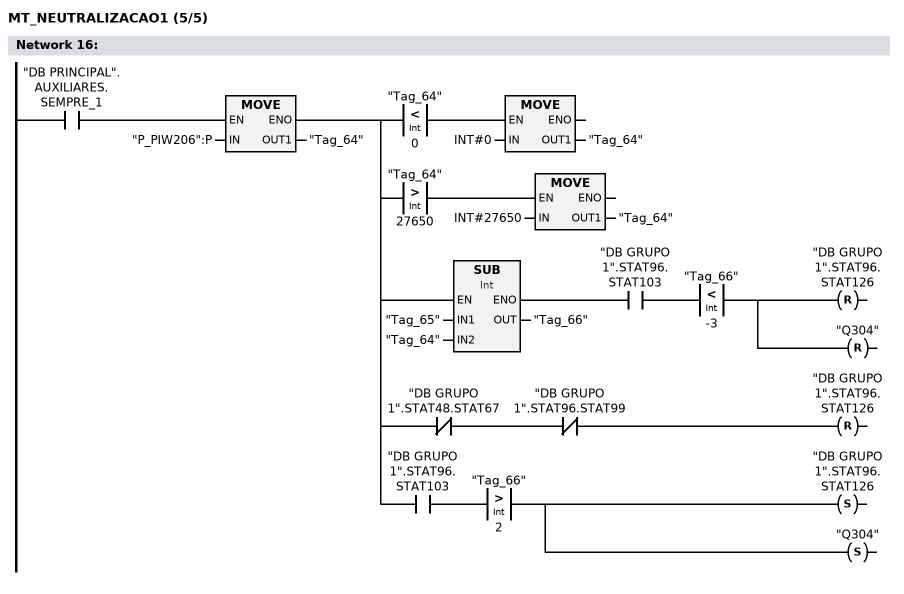
   RUNG wire#powerrail
      Contact( "DB PRINCIPAL".AUXILIARES.SEMPRE_1 )
      { S7_GenerateENO := "TRUE" } Move(in := "P_PIW206":P, out1 => "Tag_64")
      wire#w1
      { S7_Templates := "SrcType := Int" } LT_Contact(in1 := "Tag_64", in2 := 0)
      { S7_GenerateENO := "TRUE" } Move(in := INT#0, out1 => "Tag_64")
   END_RUNG
   RUNG wire#w1
      { S7_Templates := "SrcType := Int" } GT_Contact(in1 := "Tag_64", in2 := 27650)
      { S7_GenerateENO := "TRUE" } Move(in := INT#27650, out1 => "Tag_64")
   END_RUNG
   RUNG wire#w1
      { S7_Templates := "SrcType := Int"; S7_GenerateENO := "TRUE" } Sub(in1 := "Tag_65", in2 := "Tag_64", out => "Tag_66")
      Contact( "DB GRUPO 1".STAT96.STAT103 )
      { S7_Templates := "SrcType := Int" } LT_Contact(in1 := "Tag_66", in2 := -3)
      wire#w2
      R_Coil( "DB GRUPO 1".STAT96.STAT126 )
   END_RUNG
   RUNG wire#w2
      R_Coil( "Q304" )
   END_RUNG
   RUNG wire#w1
      I_Contact( "DB GRUPO 1".STAT48.STAT67 )
      I_Contact( "DB GRUPO 1".STAT96.STAT99 )
      R_Coil( "DB GRUPO 1".STAT96.STAT126 )
   END_RUNG
   RUNG wire#w1
      Contact( "DB GRUPO 1".STAT96.STAT103 )
      { S7_Templates := "SrcType := Int" } GT_Contact(in1 := "Tag_66", in2 := 2)
      wire#w3
      S_Coil( "DB GRUPO 1".STAT96.STAT126 )
   END_RUNG
   RUNG wire#w3
      S_Coil( "Q304" )
   END_RUNG
   // the same network as SCL:
   // ENO of a box is taken as its EN; it also drops when the box reports an error
   IF "DB PRINCIPAL".AUXILIARES.SEMPRE_1 THEN "Tag_64" := "P_PIW206":P; END_IF;
   IF "DB PRINCIPAL".AUXILIARES.SEMPRE_1 AND ("Tag_64" < 0) THEN "Tag_64" := INT#0; END_IF;
   IF "DB PRINCIPAL".AUXILIARES.SEMPRE_1 AND ("Tag_64" > 27650) THEN "Tag_64" := INT#27650; END_IF;
   IF "DB PRINCIPAL".AUXILIARES.SEMPRE_1 THEN "Tag_66" := "Tag_65" - "Tag_64"; END_IF;
   IF "DB PRINCIPAL".AUXILIARES.SEMPRE_1 AND "DB GRUPO 1".STAT96.STAT103 AND ("Tag_66" < (-3)) THEN
       "DB GRUPO 1".STAT96.STAT126 := FALSE;
       "Q304" := FALSE;
   END_IF;
   IF "DB PRINCIPAL".AUXILIARES.SEMPRE_1 AND NOT "DB GRUPO 1".STAT48.STAT67 AND NOT "DB GRUPO 1".STAT96.STAT99 THEN
       "DB GRUPO 1".STAT96.STAT126 := FALSE;
   END_IF;
   IF "DB PRINCIPAL".AUXILIARES.SEMPRE_1 AND "DB GRUPO 1".STAT96.STAT103 AND ("Tag_66" > 2) THEN
       "DB GRUPO 1".STAT96.STAT126 := TRUE;
       "Q304" := TRUE;
   END_IF;
END_REGION
END_FUNCTION

FUNCTION "MT_EXTRACTA1" : Void   // FC13, LAD
TITLE = MÓDULO DE CONTROLE DA EXTRACTA 1
{ S7_Optimized_Access := 'FALSE' }
AUTHOR : THALLES
FAMILY : TRAÇÃO
NAME : LINHA1
VERSION : 0.1
// DATA BLOCK DE CONTROLE // DB13
// Automation Pack Automação Indl. e Com. Ltda.
// Cliente: Texima S/A Ind. de Máquinas
// Cliente Final: Cia. Fiação e Tecidos Santo Antonio.
// Máquina: Sanforizadeira SMT-15 - O.S.: 24.626
   VAR_TEMP
      AUX_R : Real;
   END_VAR
   VAR_TEMP   // added for the SCL form of the ladder/FBD networks
      _w1 : Bool;
      _w2 : Bool;
   END_VAR
BEGIN

REGION Network 1: ALARMES
   // RESET DOS ALARMES
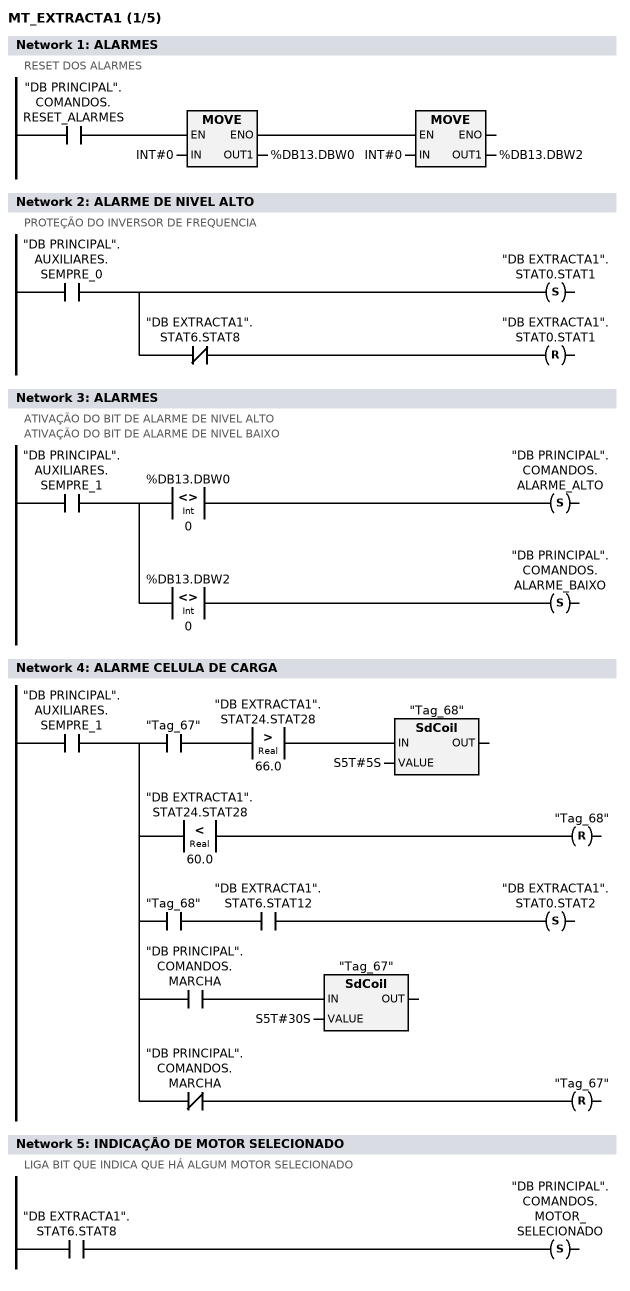
   RUNG wire#powerrail
      Contact( "DB PRINCIPAL".COMANDOS.RESET_ALARMES )
      { S7_GenerateENO := "TRUE" } Move(in := INT#0, out1 => %DB13.DBW0)
      { S7_GenerateENO := "TRUE" } Move(in := INT#0, out1 => %DB13.DBW2)
   END_RUNG
   // the same network as SCL:
   // ENO of a box is taken as its EN; it also drops when the box reports an error
   IF "DB PRINCIPAL".COMANDOS.RESET_ALARMES THEN
       %DB13.DBW0 := INT#0;
       %DB13.DBW2 := INT#0;
   END_IF;
END_REGION

REGION Network 2: ALARME DE NIVEL ALTO
   // PROTEÇÃO DO INVERSOR DE FREQUENCIA
   RUNG wire#powerrail
      Contact( "DB PRINCIPAL".AUXILIARES.SEMPRE_0 )
      wire#w1
      S_Coil( "DB EXTRACTA1".STAT0.STAT1 )
   END_RUNG
   RUNG wire#w1
      I_Contact( "DB EXTRACTA1".STAT6.STAT8 )
      R_Coil( "DB EXTRACTA1".STAT0.STAT1 )
   END_RUNG
   // the same network as SCL:
   IF "DB PRINCIPAL".AUXILIARES.SEMPRE_0 THEN "DB EXTRACTA1".STAT0.STAT1 := TRUE; END_IF;
   IF "DB PRINCIPAL".AUXILIARES.SEMPRE_0 AND NOT "DB EXTRACTA1".STAT6.STAT8 THEN
       "DB EXTRACTA1".STAT0.STAT1 := FALSE;
   END_IF;
END_REGION

REGION Network 3: ALARMES
   // ATIVAÇÃO DO BIT DE ALARME DE NIVEL ALTO
   // ATIVAÇÃO DO BIT DE ALARME DE NIVEL BAIXO
   RUNG wire#powerrail
      Contact( "DB PRINCIPAL".AUXILIARES.SEMPRE_1 )
      wire#w1
      { S7_Templates := "SrcType := Int" } NE_Contact(in1 := %DB13.DBW0, in2 := 0)
      S_Coil( "DB PRINCIPAL".COMANDOS.ALARME_ALTO )
   END_RUNG
   RUNG wire#w1
      { S7_Templates := "SrcType := Int" } NE_Contact(in1 := %DB13.DBW2, in2 := 0)
      S_Coil( "DB PRINCIPAL".COMANDOS.ALARME_BAIXO )
   END_RUNG
   // the same network as SCL:
   IF "DB PRINCIPAL".AUXILIARES.SEMPRE_1 AND (%DB13.DBW0 <> 0) THEN
       "DB PRINCIPAL".COMANDOS.ALARME_ALTO := TRUE;
   END_IF;
   IF "DB PRINCIPAL".AUXILIARES.SEMPRE_1 AND (%DB13.DBW2 <> 0) THEN
       "DB PRINCIPAL".COMANDOS.ALARME_BAIXO := TRUE;
   END_IF;
END_REGION

REGION Network 4: ALARME CELULA DE CARGA
   // no SCL statement known for SdCoil: written as a call
   #_w1 := "DB PRINCIPAL".AUXILIARES.SEMPRE_1;
   SdCoil(value := S5T#5S,
          in := "DB PRINCIPAL".AUXILIARES.SEMPRE_1 AND "Tag_67" AND ("DB EXTRACTA1".STAT24.STAT28 > 66.0),
          operand := "Tag_68");
   IF #_w1 AND ("DB EXTRACTA1".STAT24.STAT28 < 60.0) THEN "Tag_68" := FALSE; END_IF;
   IF #_w1 AND "Tag_68" AND "DB EXTRACTA1".STAT6.STAT12 THEN "DB EXTRACTA1".STAT0.STAT2 := TRUE; END_IF;
   SdCoil(value := S5T#30S, operand := "Tag_67", in := #_w1 AND "DB PRINCIPAL".COMANDOS.MARCHA);
   IF #_w1 AND NOT "DB PRINCIPAL".COMANDOS.MARCHA THEN "Tag_67" := FALSE; END_IF;
END_REGION

REGION Network 5: INDICAÇÃO DE MOTOR SELECIONADO
   // LIGA BIT QUE INDICA QUE HÁ ALGUM MOTOR SELECIONADO
   RUNG wire#powerrail
      Contact( "DB EXTRACTA1".STAT6.STAT8 )
      S_Coil( "DB PRINCIPAL".COMANDOS.MOTOR_SELECIONADO )
   END_RUNG
   // the same network as SCL:
   IF "DB EXTRACTA1".STAT6.STAT8 THEN "DB PRINCIPAL".COMANDOS.MOTOR_SELECIONADO := TRUE; END_IF;
END_REGION

REGION Network 6: COMANDO PARA SELEÇÃO DO MOTOR
   // COMANDO PARA SELEÇÃO DO MOTOR
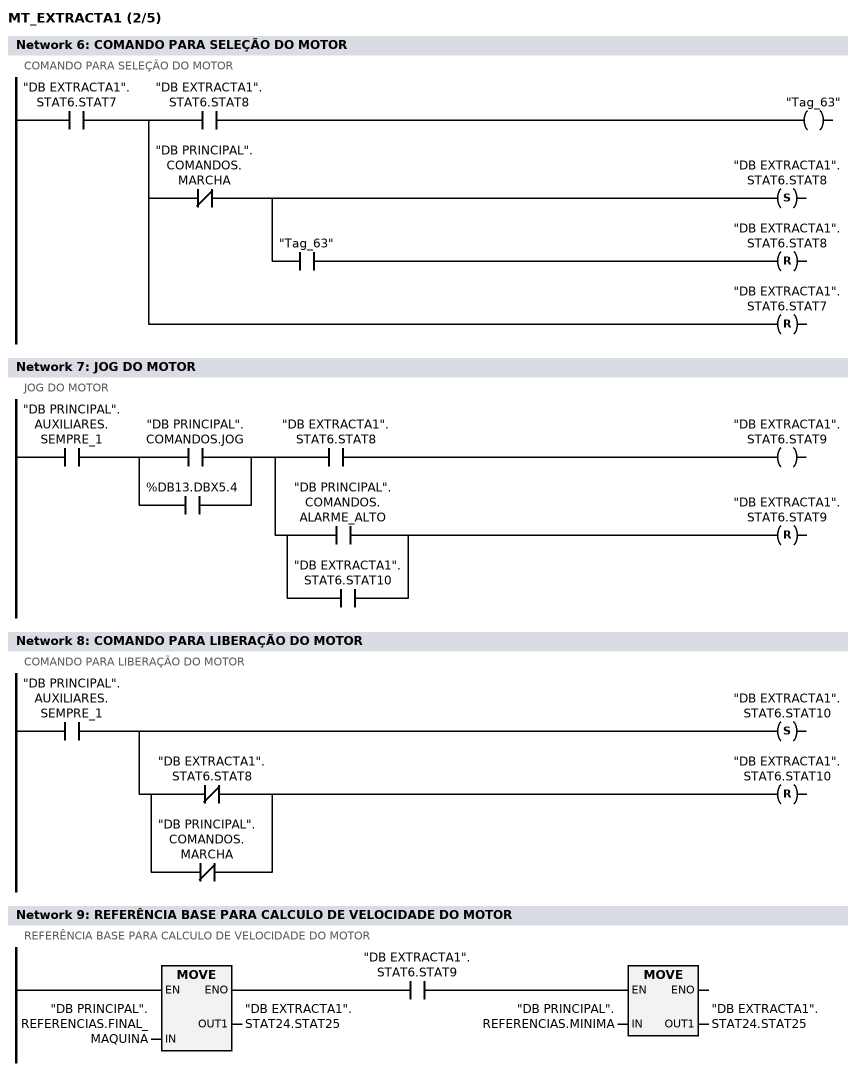
   RUNG wire#powerrail
      Contact( "DB EXTRACTA1".STAT6.STAT7 )
      wire#w1
      Contact( "DB EXTRACTA1".STAT6.STAT8 )
      Coil( "Tag_63" )
   END_RUNG
   RUNG wire#w1
      I_Contact( "DB PRINCIPAL".COMANDOS.MARCHA )
      wire#w2
      S_Coil( "DB EXTRACTA1".STAT6.STAT8 )
   END_RUNG
   RUNG wire#w2
      Contact( "Tag_63" )
      R_Coil( "DB EXTRACTA1".STAT6.STAT8 )
   END_RUNG
   RUNG wire#w1
      R_Coil( "DB EXTRACTA1".STAT6.STAT7 )
   END_RUNG
   // the same network as SCL:
   "Tag_63" := "DB EXTRACTA1".STAT6.STAT7 AND "DB EXTRACTA1".STAT6.STAT8;
   #_w1 := "DB EXTRACTA1".STAT6.STAT7 AND NOT "DB PRINCIPAL".COMANDOS.MARCHA;
   IF #_w1 THEN "DB EXTRACTA1".STAT6.STAT8 := TRUE; END_IF;
   IF #_w1 AND "Tag_63" THEN "DB EXTRACTA1".STAT6.STAT8 := FALSE; END_IF;
   IF "DB EXTRACTA1".STAT6.STAT7 THEN "DB EXTRACTA1".STAT6.STAT7 := FALSE; END_IF;
END_REGION

REGION Network 7: JOG DO MOTOR
   // JOG DO MOTOR
   RUNG wire#powerrail
      Contact( "DB PRINCIPAL".AUXILIARES.SEMPRE_1 )
      wire#w1
      Contact( "DB PRINCIPAL".COMANDOS.JOG )
      wire#w2
      Contact( "DB EXTRACTA1".STAT6.STAT8 )
      Coil( "DB EXTRACTA1".STAT6.STAT9 )
   END_RUNG
   RUNG wire#w1
      Contact( %DB13.DBX5.4 )
   END_RUNG wire#w2
   RUNG wire#w2
      Contact( "DB PRINCIPAL".COMANDOS.ALARME_ALTO )
      wire#w3
      R_Coil( "DB EXTRACTA1".STAT6.STAT9 )
   END_RUNG
   RUNG wire#w2
      Contact( "DB EXTRACTA1".STAT6.STAT10 )
   END_RUNG wire#w3
   // the same network as SCL:
   #_w1 := "DB PRINCIPAL".AUXILIARES.SEMPRE_1 AND ("DB PRINCIPAL".COMANDOS.JOG OR %DB13.DBX5.4);
   "DB EXTRACTA1".STAT6.STAT9 := #_w1 AND "DB EXTRACTA1".STAT6.STAT8;
   IF #_w1 AND ("DB PRINCIPAL".COMANDOS.ALARME_ALTO OR "DB EXTRACTA1".STAT6.STAT10) THEN
       "DB EXTRACTA1".STAT6.STAT9 := FALSE;
   END_IF;
END_REGION

REGION Network 8: COMANDO PARA LIBERAÇÃO DO MOTOR
   // COMANDO PARA LIBERAÇÃO DO MOTOR
   RUNG wire#powerrail
      Contact( "DB PRINCIPAL".AUXILIARES.SEMPRE_1 )
      wire#w1
      S_Coil( "DB EXTRACTA1".STAT6.STAT10 )
   END_RUNG
   RUNG wire#w1
      I_Contact( "DB EXTRACTA1".STAT6.STAT8 )
      wire#w2
      R_Coil( "DB EXTRACTA1".STAT6.STAT10 )
   END_RUNG
   RUNG wire#w1
      I_Contact( "DB PRINCIPAL".COMANDOS.MARCHA )
   END_RUNG wire#w2
   // the same network as SCL:
   IF "DB PRINCIPAL".AUXILIARES.SEMPRE_1 THEN "DB EXTRACTA1".STAT6.STAT10 := TRUE; END_IF;
   IF "DB PRINCIPAL".AUXILIARES.SEMPRE_1 AND (NOT "DB EXTRACTA1".STAT6.STAT8 OR NOT "DB PRINCIPAL".COMANDOS.MARCHA) THEN
       "DB EXTRACTA1".STAT6.STAT10 := FALSE;
   END_IF;
END_REGION

REGION Network 9: REFERÊNCIA BASE PARA CALCULO DE VELOCIDADE DO MOTOR
   // REFERÊNCIA BASE PARA CALCULO DE VELOCIDADE DO MOTOR
   RUNG wire#powerrail
      { S7_GenerateENO := "TRUE" } Move(in := "DB PRINCIPAL".REFERENCIAS.FINAL_MAQUINA, out1 => "DB EXTRACTA1".STAT24.STAT25)
      Contact( "DB EXTRACTA1".STAT6.STAT9 )
      { S7_GenerateENO := "TRUE" } Move(in := "DB PRINCIPAL".REFERENCIAS.MINIMA, out1 => "DB EXTRACTA1".STAT24.STAT25)
   END_RUNG
   // the same network as SCL:
   // ENO of a box is taken as its EN; it also drops when the box reports an error
   "DB EXTRACTA1".STAT24.STAT25 := "DB PRINCIPAL".REFERENCIAS.FINAL_MAQUINA;
   IF "DB EXTRACTA1".STAT6.STAT9 THEN
       "DB EXTRACTA1".STAT24.STAT25 := "DB PRINCIPAL".REFERENCIAS.MINIMA;
   END_IF;
END_REGION

REGION Network 10
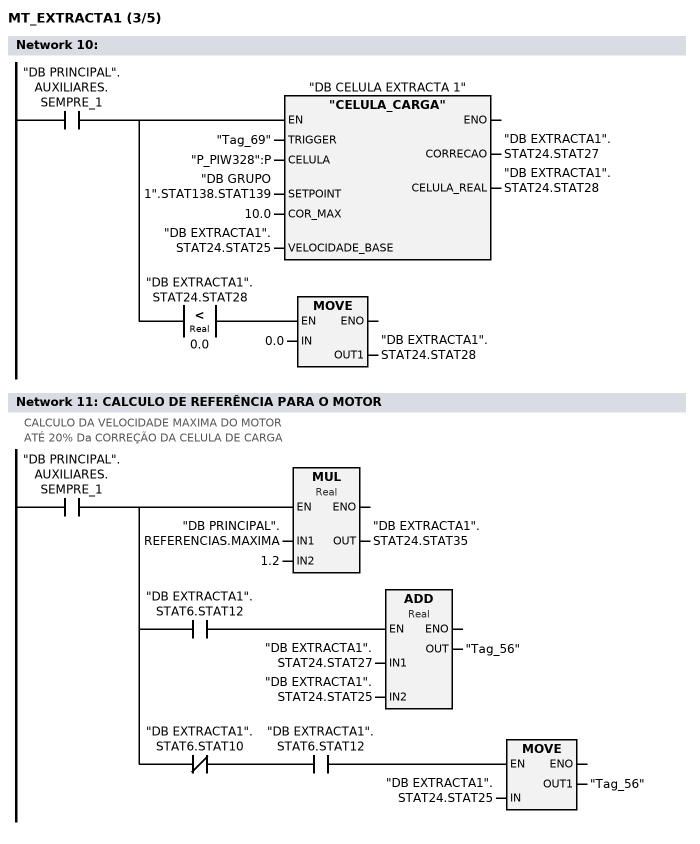
   RUNG wire#powerrail
      Contact( "DB PRINCIPAL".AUXILIARES.SEMPRE_1 )
      wire#w1
      "DB CELULA EXTRACTA 1"(TRIGGER := "Tag_69", CELULA := "P_PIW328":P, SETPOINT := "DB GRUPO 1".STAT138.STAT139, COR_MAX := 10.0, VELOCIDADE_BASE := "DB EXTRACTA1".STAT24.STAT25, CORRECAO => "DB EXTRACTA1".STAT24.STAT27, CELULA_REAL => "DB EXTRACTA1".STAT24.STAT28)
   END_RUNG
   RUNG wire#w1
      { S7_Templates := "SrcType := Real" } LT_Contact(in1 := "DB EXTRACTA1".STAT24.STAT28, in2 := 0.0)
      { S7_GenerateENO := "TRUE" } Move(in := 0.0, out1 => "DB EXTRACTA1".STAT24.STAT28)
   END_RUNG
   // the same network as SCL:
   #_w1 := "DB PRINCIPAL".AUXILIARES.SEMPRE_1;
   IF #_w1 THEN
       "DB CELULA EXTRACTA 1"(TRIGGER := "Tag_69",   // "CELULA_CARGA"
                              CELULA := "P_PIW328":P,
                              SETPOINT := "DB GRUPO 1".STAT138.STAT139,
                              COR_MAX := 10.0,
                              VELOCIDADE_BASE := "DB EXTRACTA1".STAT24.STAT25,
                              CORRECAO => "DB EXTRACTA1".STAT24.STAT27,
                              CELULA_REAL => "DB EXTRACTA1".STAT24.STAT28);
   END_IF;
   IF #_w1 AND ("DB EXTRACTA1".STAT24.STAT28 < 0.0) THEN "DB EXTRACTA1".STAT24.STAT28 := 0.0; END_IF;
END_REGION

REGION Network 11: CALCULO DE REFERÊNCIA PARA O MOTOR
   // CALCULO DA VELOCIDADE MAXIMA DO MOTOR
   // ATÉ 20% Da CORREÇÃO DA CELULA DE CARGA
   RUNG wire#powerrail
      Contact( "DB PRINCIPAL".AUXILIARES.SEMPRE_1 )
      wire#w1
      { S7_Templates := "SrcType := Real"; S7_GenerateENO := "TRUE" } Mul(in1 := "DB PRINCIPAL".REFERENCIAS.MAXIMA, in2 := 1.2, out => "DB EXTRACTA1".STAT24.STAT35)
   END_RUNG
   RUNG wire#w1
      Contact( "DB EXTRACTA1".STAT6.STAT12 )
      { S7_Templates := "SrcType := Real"; S7_GenerateENO := "TRUE" } Add(in1 := "DB EXTRACTA1".STAT24.STAT27, in2 := "DB EXTRACTA1".STAT24.STAT25, out => "Tag_56")
   END_RUNG
   RUNG wire#w1
      I_Contact( "DB EXTRACTA1".STAT6.STAT10 )
      Contact( "DB EXTRACTA1".STAT6.STAT12 )
      { S7_GenerateENO := "TRUE" } Move(in := "DB EXTRACTA1".STAT24.STAT25, out1 => "Tag_56")
   END_RUNG
   // the same network as SCL:
   IF "DB PRINCIPAL".AUXILIARES.SEMPRE_1 THEN
       "DB EXTRACTA1".STAT24.STAT35 := "DB PRINCIPAL".REFERENCIAS.MAXIMA * 1.2;
   END_IF;
   IF "DB PRINCIPAL".AUXILIARES.SEMPRE_1 AND "DB EXTRACTA1".STAT6.STAT12 THEN
       "Tag_56" := "DB EXTRACTA1".STAT24.STAT27 + "DB EXTRACTA1".STAT24.STAT25;
   END_IF;
   IF "DB PRINCIPAL".AUXILIARES.SEMPRE_1 AND NOT "DB EXTRACTA1".STAT6.STAT10 AND "DB EXTRACTA1".STAT6.STAT12 THEN
       "Tag_56" := "DB EXTRACTA1".STAT24.STAT25;
   END_IF;
END_REGION

REGION Network 12: ACC/DEC DA REFERÊNCIA DO MOTOR
   // ACC/DEC DA REFERÊNCIA DO MOTOR
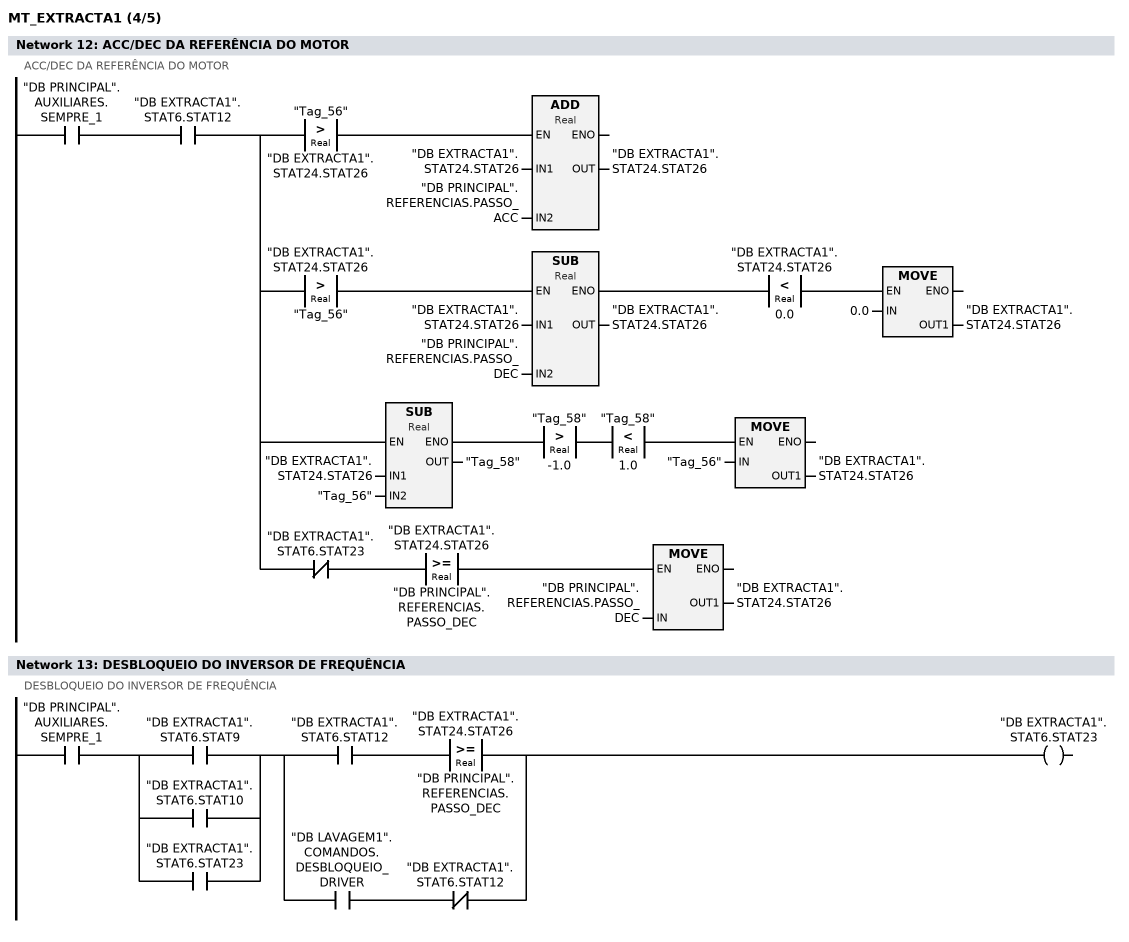
   RUNG wire#powerrail
      Contact( "DB PRINCIPAL".AUXILIARES.SEMPRE_1 )
      Contact( "DB EXTRACTA1".STAT6.STAT12 )
      wire#w1
      { S7_Templates := "SrcType := Real" } GT_Contact(in1 := "Tag_56", in2 := "DB EXTRACTA1".STAT24.STAT26)
      { S7_Templates := "SrcType := Real"; S7_GenerateENO := "TRUE" } Add(in1 := "DB EXTRACTA1".STAT24.STAT26, in2 := "DB PRINCIPAL".REFERENCIAS.PASSO_ACC, out => "DB EXTRACTA1".STAT24.STAT26)
   END_RUNG
   RUNG wire#w1
      { S7_Templates := "SrcType := Real" } GT_Contact(in1 := "DB EXTRACTA1".STAT24.STAT26, in2 := "Tag_56")
      { S7_Templates := "SrcType := Real"; S7_GenerateENO := "TRUE" } Sub(in1 := "DB EXTRACTA1".STAT24.STAT26, in2 := "DB PRINCIPAL".REFERENCIAS.PASSO_DEC, out => "DB EXTRACTA1".STAT24.STAT26)
      { S7_Templates := "SrcType := Real" } LT_Contact(in1 := "DB EXTRACTA1".STAT24.STAT26, in2 := 0.0)
      { S7_GenerateENO := "TRUE" } Move(in := 0.0, out1 => "DB EXTRACTA1".STAT24.STAT26)
   END_RUNG
   RUNG wire#w1
      { S7_Templates := "SrcType := Real"; S7_GenerateENO := "TRUE" } Sub(in1 := "DB EXTRACTA1".STAT24.STAT26, in2 := "Tag_56", out => "Tag_58")
      { S7_Templates := "SrcType := Real" } GT_Contact(in1 := "Tag_58", in2 := -1.0)
      { S7_Templates := "SrcType := Real" } LT_Contact(in1 := "Tag_58", in2 := 1.0)
      { S7_GenerateENO := "TRUE" } Move(in := "Tag_56", out1 => "DB EXTRACTA1".STAT24.STAT26)
   END_RUNG
   RUNG wire#w1
      I_Contact( "DB EXTRACTA1".STAT6.STAT23 )
      { S7_Templates := "SrcType := Real" } GE_Contact(in1 := "DB EXTRACTA1".STAT24.STAT26, in2 := "DB PRINCIPAL".REFERENCIAS.PASSO_DEC)
      { S7_GenerateENO := "TRUE" } Move(in := "DB PRINCIPAL".REFERENCIAS.PASSO_DEC, out1 => "DB EXTRACTA1".STAT24.STAT26)
   END_RUNG
   // the same network as SCL:
   // ENO of a box is taken as its EN; it also drops when the box reports an error
   #_w1 := "DB PRINCIPAL".AUXILIARES.SEMPRE_1 AND "DB EXTRACTA1".STAT6.STAT12;
   IF #_w1 AND ("Tag_56" > "DB EXTRACTA1".STAT24.STAT26) THEN
       "DB EXTRACTA1".STAT24.STAT26 := "DB EXTRACTA1".STAT24.STAT26 + "DB PRINCIPAL".REFERENCIAS.PASSO_ACC;
   END_IF;
   #_w2 := #_w1 AND ("DB EXTRACTA1".STAT24.STAT26 > "Tag_56");
   IF #_w2 THEN
       "DB EXTRACTA1".STAT24.STAT26 := "DB EXTRACTA1".STAT24.STAT26 - "DB PRINCIPAL".REFERENCIAS.PASSO_DEC;
   END_IF;
   IF #_w2 AND ("DB EXTRACTA1".STAT24.STAT26 < 0.0) THEN "DB EXTRACTA1".STAT24.STAT26 := 0.0; END_IF;
   IF #_w1 THEN "Tag_58" := "DB EXTRACTA1".STAT24.STAT26 - "Tag_56"; END_IF;
   IF #_w1 AND ("Tag_58" > (-1.0)) AND ("Tag_58" < 1.0) THEN
       "DB EXTRACTA1".STAT24.STAT26 := "Tag_56";
   END_IF;
   IF #_w1 AND NOT "DB EXTRACTA1".STAT6.STAT23 AND ("DB EXTRACTA1".STAT24.STAT26 >= "DB PRINCIPAL".REFERENCIAS.PASSO_DEC) THEN
       "DB EXTRACTA1".STAT24.STAT26 := "DB PRINCIPAL".REFERENCIAS.PASSO_DEC;
   END_IF;
END_REGION

REGION Network 13: DESBLOQUEIO DO INVERSOR DE FREQUÊNCIA
   // DESBLOQUEIO DO INVERSOR DE FREQUÊNCIA
   RUNG wire#powerrail
      Contact( "DB PRINCIPAL".AUXILIARES.SEMPRE_1 )
      wire#w1
      Contact( "DB EXTRACTA1".STAT6.STAT9 )
      wire#w2
      Contact( "DB EXTRACTA1".STAT6.STAT12 )
      { S7_Templates := "SrcType := Real" } GE_Contact(in1 := "DB EXTRACTA1".STAT24.STAT26, in2 := "DB PRINCIPAL".REFERENCIAS.PASSO_DEC)
      wire#w3
      Coil( "DB EXTRACTA1".STAT6.STAT23 )
   END_RUNG
   RUNG wire#w1
      Contact( "DB EXTRACTA1".STAT6.STAT10 )
   END_RUNG wire#w2
   RUNG wire#w1
      Contact( "DB EXTRACTA1".STAT6.STAT23 )
   END_RUNG wire#w2
   RUNG wire#w2
      Contact( "DB LAVAGEM1".COMANDOS.DESBLOQUEIO_DRIVER )
      I_Contact( "DB EXTRACTA1".STAT6.STAT12 )
   END_RUNG wire#w3
   // the same network as SCL:
   "DB EXTRACTA1".STAT6.STAT23 := "DB PRINCIPAL".AUXILIARES.SEMPRE_1 AND ("DB EXTRACTA1".STAT6.STAT9 OR "DB EXTRACTA1".STAT6.STAT10 OR "DB EXTRACTA1".STAT6.STAT23) AND (("DB EXTRACTA1".STAT6.STAT12 AND ("DB EXTRACTA1".STAT24.STAT26 >= "DB PRINCIPAL".REFERENCIAS.PASSO_DEC)) OR ("DB LAVAGEM1".COMANDOS.DESBLOQUEIO_DRIVER AND NOT "DB EXTRACTA1".STAT6.STAT12));
END_REGION

REGION Network 14
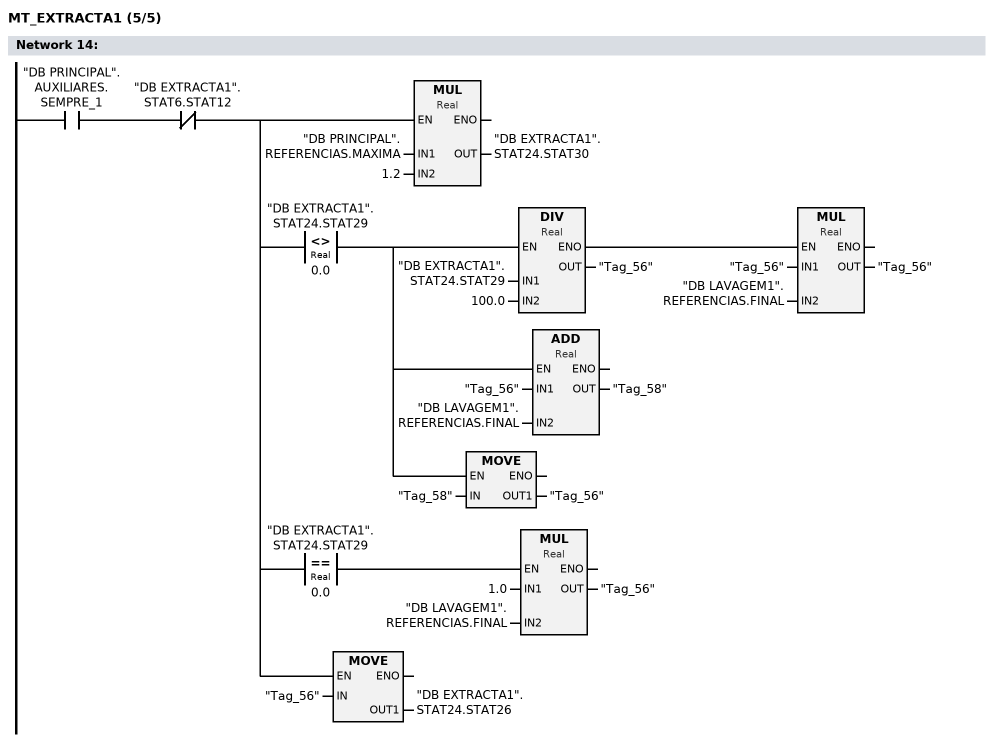
   RUNG wire#powerrail
      Contact( "DB PRINCIPAL".AUXILIARES.SEMPRE_1 )
      I_Contact( "DB EXTRACTA1".STAT6.STAT12 )
      wire#w1
      { S7_Templates := "SrcType := Real"; S7_GenerateENO := "TRUE" } Mul(in1 := "DB PRINCIPAL".REFERENCIAS.MAXIMA, in2 := 1.2, out => "DB EXTRACTA1".STAT24.STAT30)
   END_RUNG
   RUNG wire#w1
      { S7_Templates := "SrcType := Real" } NE_Contact(in1 := "DB EXTRACTA1".STAT24.STAT29, in2 := 0.0)
      wire#w2
      { S7_Templates := "SrcType := Real"; S7_GenerateENO := "TRUE" } Div(in1 := "DB EXTRACTA1".STAT24.STAT29, in2 := 100.0, out => "Tag_56")
      { S7_Templates := "SrcType := Real"; S7_GenerateENO := "TRUE" } Mul(in1 := "Tag_56", in2 := "DB LAVAGEM1".REFERENCIAS.FINAL, out => "Tag_56")
   END_RUNG
   RUNG wire#w2
      { S7_Templates := "SrcType := Real"; S7_GenerateENO := "TRUE" } Add(in1 := "Tag_56", in2 := "DB LAVAGEM1".REFERENCIAS.FINAL, out => "Tag_58")
   END_RUNG
   RUNG wire#w2
      { S7_GenerateENO := "TRUE" } Move(in := "Tag_58", out1 => "Tag_56")
   END_RUNG
   RUNG wire#w1
      { S7_Templates := "SrcType := Real" } EQ_Contact(in1 := "DB EXTRACTA1".STAT24.STAT29, in2 := 0.0)
      { S7_Templates := "SrcType := Real"; S7_GenerateENO := "TRUE" } Mul(in1 := 1.0, in2 := "DB LAVAGEM1".REFERENCIAS.FINAL, out => "Tag_56")
   END_RUNG
   RUNG wire#w1
      { S7_GenerateENO := "TRUE" } Move(in := "Tag_56", out1 => "DB EXTRACTA1".STAT24.STAT26)
   END_RUNG
   // the same network as SCL:
   // ENO of a box is taken as its EN; it also drops when the box reports an error
   #_w1 := "DB PRINCIPAL".AUXILIARES.SEMPRE_1 AND NOT "DB EXTRACTA1".STAT6.STAT12;
   IF #_w1 THEN "DB EXTRACTA1".STAT24.STAT30 := "DB PRINCIPAL".REFERENCIAS.MAXIMA * 1.2; END_IF;
   IF #_w1 AND ("DB EXTRACTA1".STAT24.STAT29 <> 0.0) THEN
       "Tag_56" := "DB EXTRACTA1".STAT24.STAT29 / 100.0;
       "Tag_56" := "Tag_56" * "DB LAVAGEM1".REFERENCIAS.FINAL;
       "Tag_58" := "Tag_56" + "DB LAVAGEM1".REFERENCIAS.FINAL;
       "Tag_56" := "Tag_58";
   END_IF;
   IF #_w1 AND ("DB EXTRACTA1".STAT24.STAT29 = 0.0) THEN
       "Tag_56" := 1.0 * "DB LAVAGEM1".REFERENCIAS.FINAL;
   END_IF;
   IF #_w1 THEN "DB EXTRACTA1".STAT24.STAT26 := "Tag_56"; END_IF;
END_REGION

REGION Network 15 (STL): STATUS / CONTROLE - INVERSOR DE FREQUÊNCIA
   // DANFOSS FC300 PROFIBUS - TEX24626INV001
   // STATUS DO INVERSOR DE FREQUÊNCIA
         L     "Tag_11":P;
         T     "Tag_1";
         AN    "Tag_59";
         =     "DB EXTRACTA1".STAT6.STAT22;

   // CONTROLE DO INVERSOR DE FREQUÊNCIA
         L     1150;
         T     "Tag_1";
         A     "DB EXTRACTA1".STAT6.STAT23;
         =     "Tag_60";
         A     "T2";
         AN    "DB EXTRACTA1".STAT6.STAT22;
         =     "Tag_61";
         L     "Tag_1";
         T     "Tag_12":P;

   // REFERÊNCIA PARA O INVERSOR DE FREQUÊNCIA
         L     "DB EXTRACTA1".STAT24.STAT26;
         RND;
         T     "Tag_13":P;
END_REGION

REGION Network 16 (STL): INVERSOR RESERVA
         A     "DB PRINCIPAL".AUXILIARES.SEMPRE_1;
         =     %L24.0;
         A     %L24.0;
         A(;
         L     "DB PRINCIPAL".AUXILIARES1.INVERSOR_RESERVA1;
         L     4;
         ==I;
         );
         =     %L24.1;
         A     %L24.1;
         JNB   M00f;
         L     "DB EXTRACTA1".STAT24.STAT26;
         L     3.456;
         *R;
         T     #AUX_R;
         RND;
         T     "P_QW100":P;
   M00f: NOP   0;
         A     %L24.1;
         A     "I130";
         S     "DB PRINCIPAL".ALARME.INV_RESERVA1;
         A     %L24.1;
         A     "DB EXTRACTA1".STAT6.STAT23;
         S     "Q134";
         A     %L24.1;
         AN    "DB EXTRACTA1".STAT6.STAT23;
         R     "Q134";
         A     %L24.0;
         A(;
         L     "DB PRINCIPAL".AUXILIARES1.INVERSOR_RESERVA2;
         L     4;
         ==I;
         );
         =     %L24.1;
         A     %L24.1;
         JNB   M010;
         L     "DB EXTRACTA1".STAT24.STAT26;
         L     3.456;
         *R;
         T     #AUX_R;
         RND;
         T     "P_QW102":P;
   M010: NOP   0;
         A     %L24.1;
         A     "I132";
         S     "DB PRINCIPAL".ALARME.INV_RESERVA2;
         A     %L24.1;
         A     "DB EXTRACTA1".STAT6.STAT23;
         S     "Q135";
         A     %L24.1;
         AN    "DB EXTRACTA1".STAT6.STAT23;
         R     "Q135";
END_REGION
END_FUNCTION

FUNCTION "MT_LAVAGEM1" : Void   // FC14, LAD
TITLE = MÓDULO DE CONTROLE DA LAVAGEM 1
{ S7_Optimized_Access := 'FALSE' }
AUTHOR : THALLES
FAMILY : TRAÇÃO
NAME : LINHA1
VERSION : 0.1
// DATA BLOCK DE CONTROLE // DB14
// Automation Pack Automação Indl. e Com. Ltda.
// Cliente: Texima S/A Ind. de Máquinas
// Cliente Final: Cia. Fiação e Tecidos Santo Antonio.
// Máquina: LINHA 1 DENIN - O.S.: 24.626
   VAR_TEMP
      AUX_R : Real;
   END_VAR
   VAR_TEMP   // added for the SCL form of the ladder/FBD networks
      _w1 : Bool;
   END_VAR
BEGIN

REGION Network 1: ALARMES
   // RESET DOS ALARMES
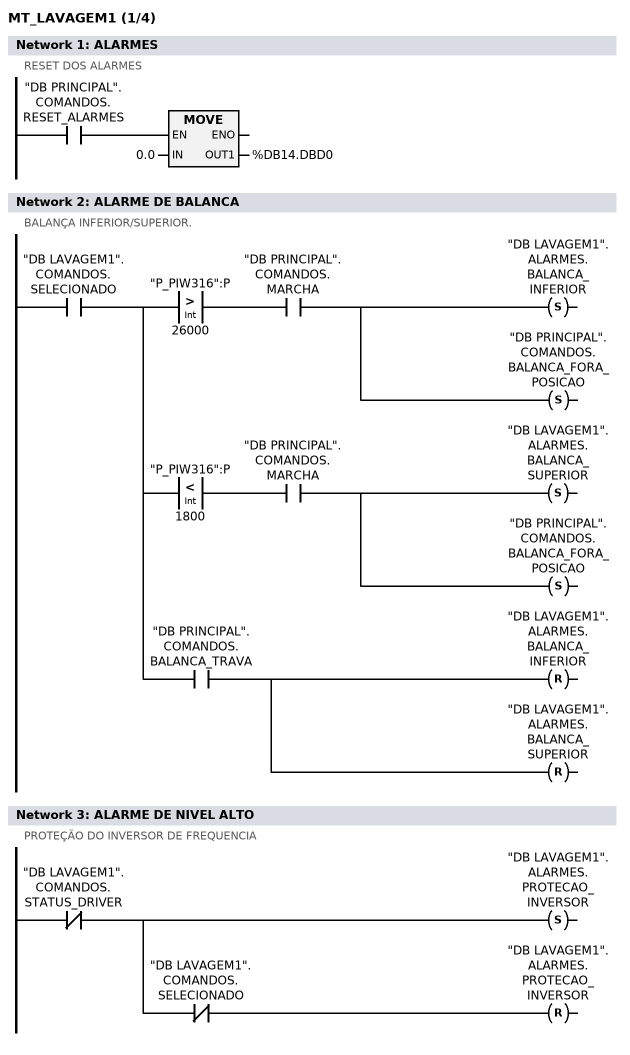
   RUNG wire#powerrail
      Contact( "DB PRINCIPAL".COMANDOS.RESET_ALARMES )
      { S7_GenerateENO := "TRUE" } Move(in := 0.0, out1 => %DB14.DBD0)
   END_RUNG
   // the same network as SCL:
   IF "DB PRINCIPAL".COMANDOS.RESET_ALARMES THEN %DB14.DBD0 := 0.0; END_IF;
END_REGION

REGION Network 2: ALARME DE BALANCA
   // BALANÇA INFERIOR/SUPERIOR.
   RUNG wire#powerrail
      Contact( "DB LAVAGEM1".COMANDOS.SELECIONADO )
      wire#w1
      { S7_Templates := "SrcType := Int" } GT_Contact(in1 := "P_PIW316":P, in2 := 26000)
      Contact( "DB PRINCIPAL".COMANDOS.MARCHA )
      wire#w2
      S_Coil( "DB LAVAGEM1".ALARMES.BALANCA_INFERIOR )
   END_RUNG
   RUNG wire#w2
      S_Coil( "DB PRINCIPAL".COMANDOS.BALANCA_FORA_POSICAO )
   END_RUNG
   RUNG wire#w1
      { S7_Templates := "SrcType := Int" } LT_Contact(in1 := "P_PIW316":P, in2 := 1800)
      Contact( "DB PRINCIPAL".COMANDOS.MARCHA )
      wire#w3
      S_Coil( "DB LAVAGEM1".ALARMES.BALANCA_SUPERIOR )
   END_RUNG
   RUNG wire#w3
      S_Coil( "DB PRINCIPAL".COMANDOS.BALANCA_FORA_POSICAO )
   END_RUNG
   RUNG wire#w1
      Contact( "DB PRINCIPAL".COMANDOS.BALANCA_TRAVA )
      wire#w4
      R_Coil( "DB LAVAGEM1".ALARMES.BALANCA_INFERIOR )
   END_RUNG
   RUNG wire#w4
      R_Coil( "DB LAVAGEM1".ALARMES.BALANCA_SUPERIOR )
   END_RUNG
   // the same network as SCL:
   IF "DB LAVAGEM1".COMANDOS.SELECIONADO AND ("P_PIW316":P > 26000) AND "DB PRINCIPAL".COMANDOS.MARCHA THEN
       "DB LAVAGEM1".ALARMES.BALANCA_INFERIOR := TRUE;
       "DB PRINCIPAL".COMANDOS.BALANCA_FORA_POSICAO := TRUE;
   END_IF;
   IF "DB LAVAGEM1".COMANDOS.SELECIONADO AND ("P_PIW316":P < 1800) AND "DB PRINCIPAL".COMANDOS.MARCHA THEN
       "DB LAVAGEM1".ALARMES.BALANCA_SUPERIOR := TRUE;
       "DB PRINCIPAL".COMANDOS.BALANCA_FORA_POSICAO := TRUE;
   END_IF;
   IF "DB LAVAGEM1".COMANDOS.SELECIONADO AND "DB PRINCIPAL".COMANDOS.BALANCA_TRAVA THEN
       "DB LAVAGEM1".ALARMES.BALANCA_INFERIOR := FALSE;
       "DB LAVAGEM1".ALARMES.BALANCA_SUPERIOR := FALSE;
   END_IF;
END_REGION

REGION Network 3: ALARME DE NIVEL ALTO
   // PROTEÇÃO DO INVERSOR DE FREQUENCIA
   RUNG wire#powerrail
      I_Contact( "DB LAVAGEM1".COMANDOS.STATUS_DRIVER )
      wire#w1
      S_Coil( "DB LAVAGEM1".ALARMES.PROTECAO_INVERSOR )
   END_RUNG
   RUNG wire#w1
      I_Contact( "DB LAVAGEM1".COMANDOS.SELECIONADO )
      R_Coil( "DB LAVAGEM1".ALARMES.PROTECAO_INVERSOR )
   END_RUNG
   // the same network as SCL:
   #_w1 := NOT "DB LAVAGEM1".COMANDOS.STATUS_DRIVER;
   IF #_w1 THEN "DB LAVAGEM1".ALARMES.PROTECAO_INVERSOR := TRUE; END_IF;
   IF #_w1 AND NOT "DB LAVAGEM1".COMANDOS.SELECIONADO THEN
       "DB LAVAGEM1".ALARMES.PROTECAO_INVERSOR := FALSE;
   END_IF;
END_REGION

REGION Network 4: ALARMES
   // ATIVAÇÃO DO BIT DE ALARME DE NIVEL ALTO
   // ATIVAÇÃO DO BIT DE ALARME DE NIVEL BAIXO
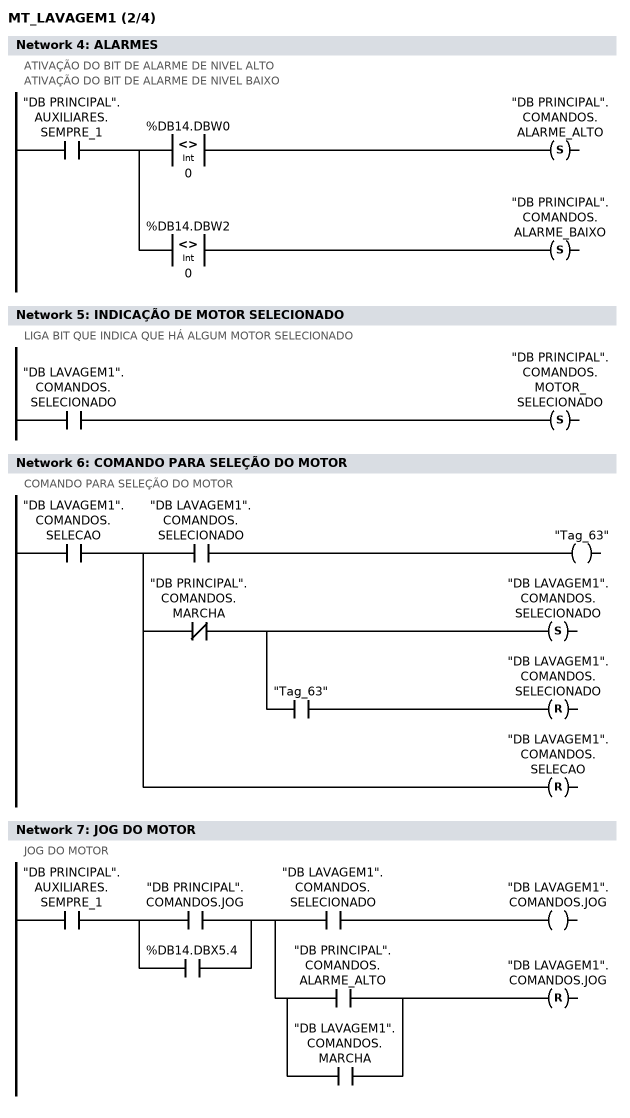
   RUNG wire#powerrail
      Contact( "DB PRINCIPAL".AUXILIARES.SEMPRE_1 )
      wire#w1
      { S7_Templates := "SrcType := Int" } NE_Contact(in1 := %DB14.DBW0, in2 := 0)
      S_Coil( "DB PRINCIPAL".COMANDOS.ALARME_ALTO )
   END_RUNG
   RUNG wire#w1
      { S7_Templates := "SrcType := Int" } NE_Contact(in1 := %DB14.DBW2, in2 := 0)
      S_Coil( "DB PRINCIPAL".COMANDOS.ALARME_BAIXO )
   END_RUNG
   // the same network as SCL:
   IF "DB PRINCIPAL".AUXILIARES.SEMPRE_1 AND (%DB14.DBW0 <> 0) THEN
       "DB PRINCIPAL".COMANDOS.ALARME_ALTO := TRUE;
   END_IF;
   IF "DB PRINCIPAL".AUXILIARES.SEMPRE_1 AND (%DB14.DBW2 <> 0) THEN
       "DB PRINCIPAL".COMANDOS.ALARME_BAIXO := TRUE;
   END_IF;
END_REGION

REGION Network 5: INDICAÇÃO DE MOTOR SELECIONADO
   // LIGA BIT QUE INDICA QUE HÁ ALGUM MOTOR SELECIONADO
   RUNG wire#powerrail
      Contact( "DB LAVAGEM1".COMANDOS.SELECIONADO )
      S_Coil( "DB PRINCIPAL".COMANDOS.MOTOR_SELECIONADO )
   END_RUNG
   // the same network as SCL:
   IF "DB LAVAGEM1".COMANDOS.SELECIONADO THEN "DB PRINCIPAL".COMANDOS.MOTOR_SELECIONADO := TRUE; END_IF;
END_REGION

REGION Network 6: COMANDO PARA SELEÇÃO DO MOTOR
   // COMANDO PARA SELEÇÃO DO MOTOR
   RUNG wire#powerrail
      Contact( "DB LAVAGEM1".COMANDOS.SELECAO )
      wire#w1
      Contact( "DB LAVAGEM1".COMANDOS.SELECIONADO )
      Coil( "Tag_63" )
   END_RUNG
   RUNG wire#w1
      I_Contact( "DB PRINCIPAL".COMANDOS.MARCHA )
      wire#w2
      S_Coil( "DB LAVAGEM1".COMANDOS.SELECIONADO )
   END_RUNG
   RUNG wire#w2
      Contact( "Tag_63" )
      R_Coil( "DB LAVAGEM1".COMANDOS.SELECIONADO )
   END_RUNG
   RUNG wire#w1
      R_Coil( "DB LAVAGEM1".COMANDOS.SELECAO )
   END_RUNG
   // the same network as SCL:
   "Tag_63" := "DB LAVAGEM1".COMANDOS.SELECAO AND "DB LAVAGEM1".COMANDOS.SELECIONADO;
   #_w1 := "DB LAVAGEM1".COMANDOS.SELECAO AND NOT "DB PRINCIPAL".COMANDOS.MARCHA;
   IF #_w1 THEN "DB LAVAGEM1".COMANDOS.SELECIONADO := TRUE; END_IF;
   IF #_w1 AND "Tag_63" THEN "DB LAVAGEM1".COMANDOS.SELECIONADO := FALSE; END_IF;
   IF "DB LAVAGEM1".COMANDOS.SELECAO THEN "DB LAVAGEM1".COMANDOS.SELECAO := FALSE; END_IF;
END_REGION

REGION Network 7: JOG DO MOTOR
   // JOG DO MOTOR
   RUNG wire#powerrail
      Contact( "DB PRINCIPAL".AUXILIARES.SEMPRE_1 )
      wire#w1
      Contact( "DB PRINCIPAL".COMANDOS.JOG )
      wire#w2
      Contact( "DB LAVAGEM1".COMANDOS.SELECIONADO )
      Coil( "DB LAVAGEM1".COMANDOS.JOG )
   END_RUNG
   RUNG wire#w1
      Contact( %DB14.DBX5.4 )
   END_RUNG wire#w2
   RUNG wire#w2
      Contact( "DB PRINCIPAL".COMANDOS.ALARME_ALTO )
      wire#w3
      R_Coil( "DB LAVAGEM1".COMANDOS.JOG )
   END_RUNG
   RUNG wire#w2
      Contact( "DB LAVAGEM1".COMANDOS.MARCHA )
   END_RUNG wire#w3
   // the same network as SCL:
   #_w1 := "DB PRINCIPAL".AUXILIARES.SEMPRE_1 AND ("DB PRINCIPAL".COMANDOS.JOG OR %DB14.DBX5.4);
   "DB LAVAGEM1".COMANDOS.JOG := #_w1 AND "DB LAVAGEM1".COMANDOS.SELECIONADO;
   IF #_w1 AND ("DB PRINCIPAL".COMANDOS.ALARME_ALTO OR "DB LAVAGEM1".COMANDOS.MARCHA) THEN
       "DB LAVAGEM1".COMANDOS.JOG := FALSE;
   END_IF;
END_REGION

REGION Network 8: COMANDO PARA LIBERAÇÃO DO MOTOR
   // COMANDO PARA LIBERAÇÃO DO MOTOR
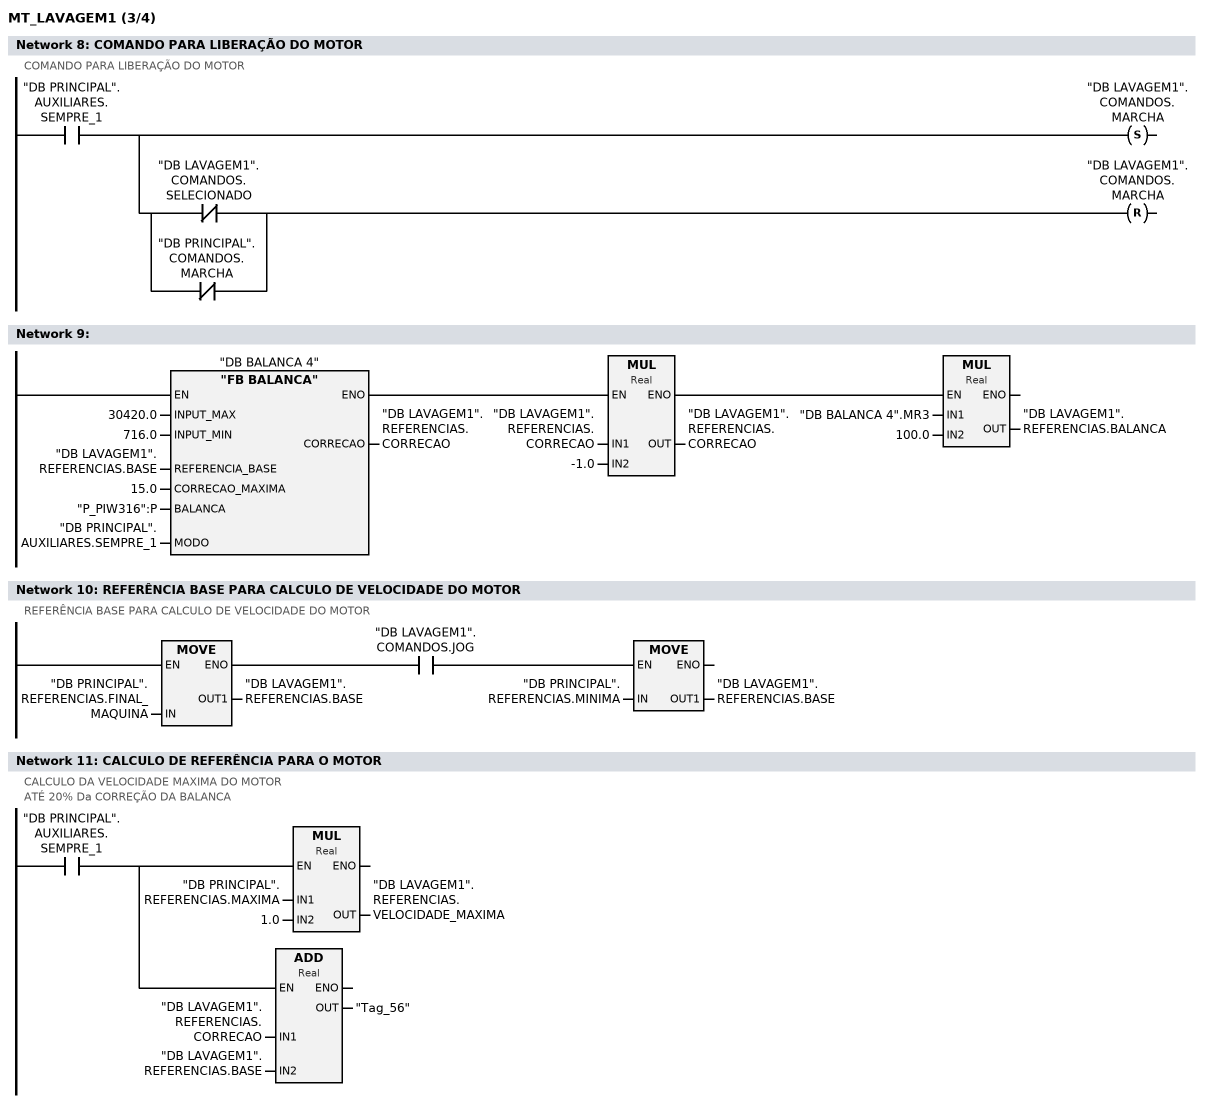
   RUNG wire#powerrail
      Contact( "DB PRINCIPAL".AUXILIARES.SEMPRE_1 )
      wire#w1
      S_Coil( "DB LAVAGEM1".COMANDOS.MARCHA )
   END_RUNG
   RUNG wire#w1
      I_Contact( "DB LAVAGEM1".COMANDOS.SELECIONADO )
      wire#w2
      R_Coil( "DB LAVAGEM1".COMANDOS.MARCHA )
   END_RUNG
   RUNG wire#w1
      I_Contact( "DB PRINCIPAL".COMANDOS.MARCHA )
   END_RUNG wire#w2
   // the same network as SCL:
   IF "DB PRINCIPAL".AUXILIARES.SEMPRE_1 THEN "DB LAVAGEM1".COMANDOS.MARCHA := TRUE; END_IF;
   IF "DB PRINCIPAL".AUXILIARES.SEMPRE_1 AND (NOT "DB LAVAGEM1".COMANDOS.SELECIONADO OR NOT "DB PRINCIPAL".COMANDOS.MARCHA) THEN
       "DB LAVAGEM1".COMANDOS.MARCHA := FALSE;
   END_IF;
END_REGION

REGION Network 9
   RUNG wire#powerrail
      "DB BALANCA 4"(INPUT_MAX := 30420.0, INPUT_MIN := 716.0, REFERENCIA_BASE := "DB LAVAGEM1".REFERENCIAS.BASE, CORRECAO_MAXIMA := 15.0, BALANCA := "P_PIW316":P, MODO := "DB PRINCIPAL".AUXILIARES.SEMPRE_1, CORRECAO => "DB LAVAGEM1".REFERENCIAS.CORRECAO)
      { S7_Templates := "SrcType := Real"; S7_GenerateENO := "TRUE" } Mul(in1 := "DB LAVAGEM1".REFERENCIAS.CORRECAO, in2 := -1.0, out => "DB LAVAGEM1".REFERENCIAS.CORRECAO)
      { S7_Templates := "SrcType := Real"; S7_GenerateENO := "TRUE" } Mul(in1 := "DB BALANCA 4".MR3, in2 := 100.0, out => "DB LAVAGEM1".REFERENCIAS.BALANCA)
   END_RUNG
   // the same network as SCL:
   // ENO of a box is taken as its EN; it also drops when the box reports an error
   "DB BALANCA 4"(INPUT_MAX := 30420.0,   // "FB BALANCA"
                  INPUT_MIN := 716.0,
                  REFERENCIA_BASE := "DB LAVAGEM1".REFERENCIAS.BASE,
                  CORRECAO_MAXIMA := 15.0,
                  BALANCA := "P_PIW316":P,
                  MODO := "DB PRINCIPAL".AUXILIARES.SEMPRE_1,
                  CORRECAO => "DB LAVAGEM1".REFERENCIAS.CORRECAO,
                  ENO => #_w1);
   IF #_w1 THEN
       "DB LAVAGEM1".REFERENCIAS.CORRECAO := "DB LAVAGEM1".REFERENCIAS.CORRECAO * (-1.0);
       "DB LAVAGEM1".REFERENCIAS.BALANCA := "DB BALANCA 4".MR3 * 100.0;
   END_IF;
END_REGION

REGION Network 10: REFERÊNCIA BASE PARA CALCULO DE VELOCIDADE DO MOTOR
   // REFERÊNCIA BASE PARA CALCULO DE VELOCIDADE DO MOTOR
   RUNG wire#powerrail
      { S7_GenerateENO := "TRUE" } Move(in := "DB PRINCIPAL".REFERENCIAS.FINAL_MAQUINA, out1 => "DB LAVAGEM1".REFERENCIAS.BASE)
      Contact( "DB LAVAGEM1".COMANDOS.JOG )
      { S7_GenerateENO := "TRUE" } Move(in := "DB PRINCIPAL".REFERENCIAS.MINIMA, out1 => "DB LAVAGEM1".REFERENCIAS.BASE)
   END_RUNG
   // the same network as SCL:
   // ENO of a box is taken as its EN; it also drops when the box reports an error
   "DB LAVAGEM1".REFERENCIAS.BASE := "DB PRINCIPAL".REFERENCIAS.FINAL_MAQUINA;
   IF "DB LAVAGEM1".COMANDOS.JOG THEN
       "DB LAVAGEM1".REFERENCIAS.BASE := "DB PRINCIPAL".REFERENCIAS.MINIMA;
   END_IF;
END_REGION

REGION Network 11: CALCULO DE REFERÊNCIA PARA O MOTOR
   // CALCULO DA VELOCIDADE MAXIMA DO MOTOR
   // ATÉ 20% Da CORREÇÃO DA BALANCA
   RUNG wire#powerrail
      Contact( "DB PRINCIPAL".AUXILIARES.SEMPRE_1 )
      wire#w1
      { S7_Templates := "SrcType := Real"; S7_GenerateENO := "TRUE" } Mul(in1 := "DB PRINCIPAL".REFERENCIAS.MAXIMA, in2 := 1.0, out => "DB LAVAGEM1".REFERENCIAS.VELOCIDADE_MAXIMA)
   END_RUNG
   RUNG wire#w1
      { S7_Templates := "SrcType := Real"; S7_GenerateENO := "TRUE" } Add(in1 := "DB LAVAGEM1".REFERENCIAS.CORRECAO, in2 := "DB LAVAGEM1".REFERENCIAS.BASE, out => "Tag_56")
   END_RUNG
   // the same network as SCL:
   IF "DB PRINCIPAL".AUXILIARES.SEMPRE_1 THEN
       "DB LAVAGEM1".REFERENCIAS.VELOCIDADE_MAXIMA := "DB PRINCIPAL".REFERENCIAS.MAXIMA * 1.0;
       "Tag_56" := "DB LAVAGEM1".REFERENCIAS.CORRECAO + "DB LAVAGEM1".REFERENCIAS.BASE;
   END_IF;
END_REGION

REGION Network 12: ACC/DEC DA REFERÊNCIA DO MOTOR
   // ACC/DEC DA REFERÊNCIA DO MOTOR
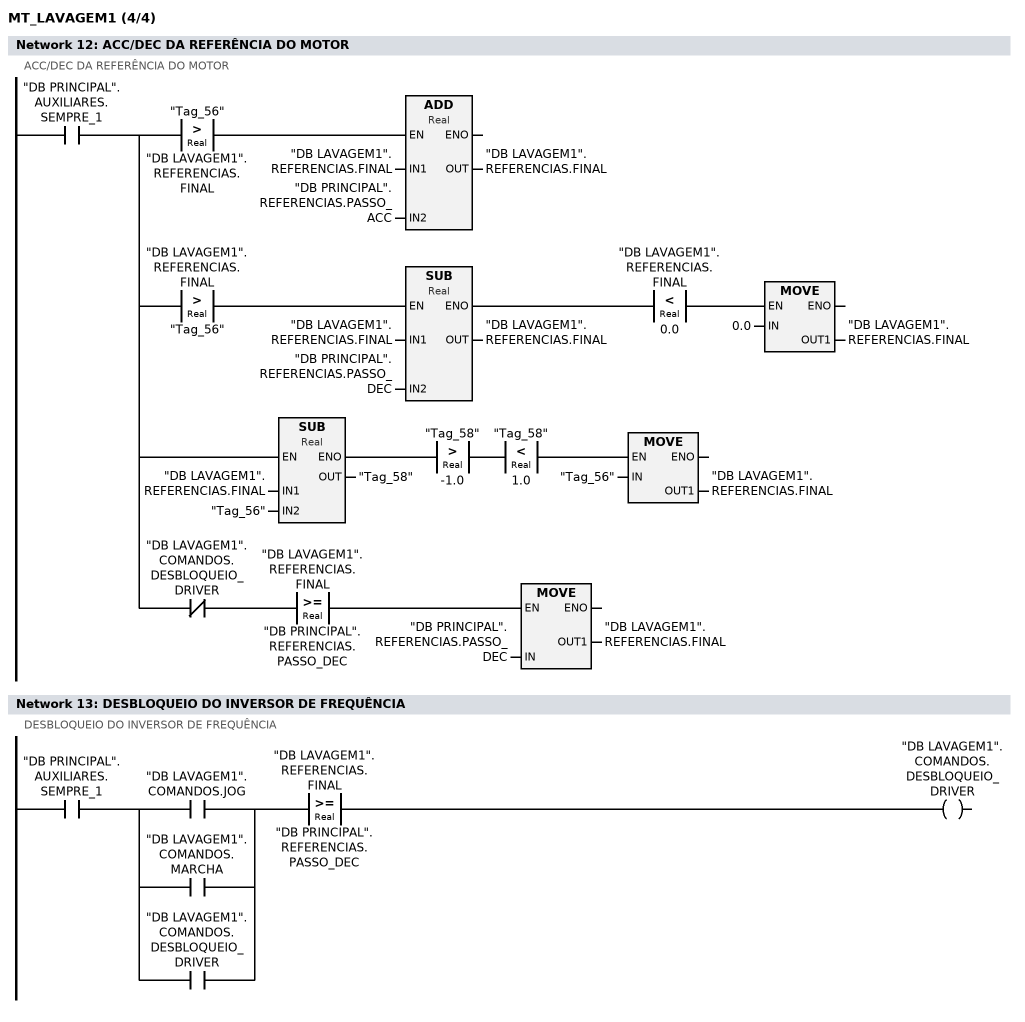
   RUNG wire#powerrail
      Contact( "DB PRINCIPAL".AUXILIARES.SEMPRE_1 )
      wire#w1
      { S7_Templates := "SrcType := Real" } GT_Contact(in1 := "Tag_56", in2 := "DB LAVAGEM1".REFERENCIAS.FINAL)
      { S7_Templates := "SrcType := Real"; S7_GenerateENO := "TRUE" } Add(in1 := "DB LAVAGEM1".REFERENCIAS.FINAL, in2 := "DB PRINCIPAL".REFERENCIAS.PASSO_ACC, out => "DB LAVAGEM1".REFERENCIAS.FINAL)
   END_RUNG
   RUNG wire#w1
      { S7_Templates := "SrcType := Real" } GT_Contact(in1 := "DB LAVAGEM1".REFERENCIAS.FINAL, in2 := "Tag_56")
      { S7_Templates := "SrcType := Real"; S7_GenerateENO := "TRUE" } Sub(in1 := "DB LAVAGEM1".REFERENCIAS.FINAL, in2 := "DB PRINCIPAL".REFERENCIAS.PASSO_DEC, out => "DB LAVAGEM1".REFERENCIAS.FINAL)
      { S7_Templates := "SrcType := Real" } LT_Contact(in1 := "DB LAVAGEM1".REFERENCIAS.FINAL, in2 := 0.0)
      { S7_GenerateENO := "TRUE" } Move(in := 0.0, out1 => "DB LAVAGEM1".REFERENCIAS.FINAL)
   END_RUNG
   RUNG wire#w1
      { S7_Templates := "SrcType := Real"; S7_GenerateENO := "TRUE" } Sub(in1 := "DB LAVAGEM1".REFERENCIAS.FINAL, in2 := "Tag_56", out => "Tag_58")
      { S7_Templates := "SrcType := Real" } GT_Contact(in1 := "Tag_58", in2 := -1.0)
      { S7_Templates := "SrcType := Real" } LT_Contact(in1 := "Tag_58", in2 := 1.0)
      { S7_GenerateENO := "TRUE" } Move(in := "Tag_56", out1 => "DB LAVAGEM1".REFERENCIAS.FINAL)
   END_RUNG
   RUNG wire#w1
      I_Contact( "DB LAVAGEM1".COMANDOS.DESBLOQUEIO_DRIVER )
      { S7_Templates := "SrcType := Real" } GE_Contact(in1 := "DB LAVAGEM1".REFERENCIAS.FINAL, in2 := "DB PRINCIPAL".REFERENCIAS.PASSO_DEC)
      { S7_GenerateENO := "TRUE" } Move(in := "DB PRINCIPAL".REFERENCIAS.PASSO_DEC, out1 => "DB LAVAGEM1".REFERENCIAS.FINAL)
   END_RUNG
   // the same network as SCL:
   // ENO of a box is taken as its EN; it also drops when the box reports an error
   IF "DB PRINCIPAL".AUXILIARES.SEMPRE_1 AND ("Tag_56" > "DB LAVAGEM1".REFERENCIAS.FINAL) THEN
       "DB LAVAGEM1".REFERENCIAS.FINAL := "DB LAVAGEM1".REFERENCIAS.FINAL + "DB PRINCIPAL".REFERENCIAS.PASSO_ACC;
   END_IF;
   #_w1 := "DB PRINCIPAL".AUXILIARES.SEMPRE_1 AND ("DB LAVAGEM1".REFERENCIAS.FINAL > "Tag_56");
   IF #_w1 THEN
       "DB LAVAGEM1".REFERENCIAS.FINAL := "DB LAVAGEM1".REFERENCIAS.FINAL - "DB PRINCIPAL".REFERENCIAS.PASSO_DEC;
   END_IF;
   IF #_w1 AND ("DB LAVAGEM1".REFERENCIAS.FINAL < 0.0) THEN "DB LAVAGEM1".REFERENCIAS.FINAL := 0.0; END_IF;
   IF "DB PRINCIPAL".AUXILIARES.SEMPRE_1 THEN "Tag_58" := "DB LAVAGEM1".REFERENCIAS.FINAL - "Tag_56"; END_IF;
   IF "DB PRINCIPAL".AUXILIARES.SEMPRE_1 AND ("Tag_58" > (-1.0)) AND ("Tag_58" < 1.0) THEN
       "DB LAVAGEM1".REFERENCIAS.FINAL := "Tag_56";
   END_IF;
   IF "DB PRINCIPAL".AUXILIARES.SEMPRE_1 AND NOT "DB LAVAGEM1".COMANDOS.DESBLOQUEIO_DRIVER AND ("DB LAVAGEM1".REFERENCIAS.FINAL >= "DB PRINCIPAL".REFERENCIAS.PASSO_DEC) THEN
       "DB LAVAGEM1".REFERENCIAS.FINAL := "DB PRINCIPAL".REFERENCIAS.PASSO_DEC;
   END_IF;
END_REGION

REGION Network 13: DESBLOQUEIO DO INVERSOR DE FREQUÊNCIA
   // DESBLOQUEIO DO INVERSOR DE FREQUÊNCIA
   RUNG wire#powerrail
      Contact( "DB PRINCIPAL".AUXILIARES.SEMPRE_1 )
      wire#w1
      Contact( "DB LAVAGEM1".COMANDOS.JOG )
      wire#w2
      { S7_Templates := "SrcType := Real" } GE_Contact(in1 := "DB LAVAGEM1".REFERENCIAS.FINAL, in2 := "DB PRINCIPAL".REFERENCIAS.PASSO_DEC)
      Coil( "DB LAVAGEM1".COMANDOS.DESBLOQUEIO_DRIVER )
   END_RUNG
   RUNG wire#w1
      Contact( "DB LAVAGEM1".COMANDOS.MARCHA )
   END_RUNG wire#w2
   RUNG wire#w1
      Contact( "DB LAVAGEM1".COMANDOS.DESBLOQUEIO_DRIVER )
   END_RUNG wire#w2
   // the same network as SCL:
   "DB LAVAGEM1".COMANDOS.DESBLOQUEIO_DRIVER := "DB PRINCIPAL".AUXILIARES.SEMPRE_1 AND ("DB LAVAGEM1".COMANDOS.JOG OR "DB LAVAGEM1".COMANDOS.MARCHA OR "DB LAVAGEM1".COMANDOS.DESBLOQUEIO_DRIVER) AND ("DB LAVAGEM1".REFERENCIAS.FINAL >= "DB PRINCIPAL".REFERENCIAS.PASSO_DEC);
END_REGION

REGION Network 14 (STL): STATUS / CONTROLE - INVERSOR DE FREQUÊNCIA
   // DANFOSS FC300 PROFIBUS - TEX24626INV001
   // STATUS DO INVERSOR DE FREQUÊNCIA
         L     "Tag_14":P;
         T     "Tag_1";
         AN    "Tag_59";
         =     "DB LAVAGEM1".COMANDOS.STATUS_DRIVER;

   // CONTROLE DO INVERSOR DE FREQUÊNCIA
         L     1150;
         T     "Tag_1";
         A     "DB LAVAGEM1".COMANDOS.DESBLOQUEIO_DRIVER;
         =     "Tag_60";
         A     "T2";
         AN    "DB LAVAGEM1".COMANDOS.STATUS_DRIVER;
         =     "Tag_61";
         L     "Tag_1";
         T     "Tag_15":P;

   // REFERÊNCIA PARA O INVERSOR DE FREQUÊNCIA
         L     "DB LAVAGEM1".REFERENCIAS.FINAL;
         L     16384.0;
         *R;

         L     "DB LAVAGEM1".REFERENCIAS.VELOCIDADE_MAXIMA;
         /R;
         RND;
         T     "Tag_62";
         L     "Tag_62";
         T     "Tag_16":P;
END_REGION

REGION Network 15 (STL): INVERSOR RESERVA
         A     "DB PRINCIPAL".AUXILIARES.SEMPRE_1;
         =     %L24.0;
         A     %L24.0;
         A(;
         L     "DB PRINCIPAL".AUXILIARES1.INVERSOR_RESERVA1;
         L     5;
         ==I;
         );
         =     %L24.1;
         A     %L24.1;
         JNB   M00d;
         L     "DB LAVAGEM1".REFERENCIAS.FINAL;
         L     3.456;
         *R;
         T     #AUX_R;
         RND;
         T     "P_QW100":P;
   M00d: NOP   0;
         A     %L24.1;
         A     "I130";
         S     "DB PRINCIPAL".ALARME.INV_RESERVA1;
         A     %L24.1;
         A     "DB LAVAGEM1".COMANDOS.DESBLOQUEIO_DRIVER;
         S     "Q134";
         A     %L24.1;
         AN    "DB LAVAGEM1".COMANDOS.DESBLOQUEIO_DRIVER;
         R     "Q134";
         A     %L24.0;
         A(;
         L     "DB PRINCIPAL".AUXILIARES1.INVERSOR_RESERVA2;
         L     5;
         ==I;
         );
         =     %L24.1;
         A     %L24.1;
         JNB   M00e;
         L     "DB LAVAGEM1".REFERENCIAS.FINAL;
         L     3.456;
         *R;
         T     #AUX_R;
         RND;
         T     "P_QW102":P;
   M00e: NOP   0;
         A     %L24.1;
         A     "I132";
         S     "DB PRINCIPAL".ALARME.INV_RESERVA2;
         A     %L24.1;
         A     "DB LAVAGEM1".COMANDOS.DESBLOQUEIO_DRIVER;
         S     "Q135";
         A     %L24.1;
         AN    "DB LAVAGEM1".COMANDOS.DESBLOQUEIO_DRIVER;
         R     "Q135";
END_REGION
END_FUNCTION

FUNCTION "MT_NEUTRALIZACAO2" : Void   // FC15, LAD
TITLE = MÓDULO DE CONTROLE DA NEUTRALIZACAO 2
{ S7_Optimized_Access := 'FALSE' }
AUTHOR : THALLES
FAMILY : TRAÇÃO
NAME : LINHA1
VERSION : 0.1
// DATA BLOCK DE CONTROLE // DB15
// Automation Pack Automação Indl. e Com. Ltda.
// Cliente: Texima S/A Ind. de Máquinas
// Cliente Final: Cia. Fiação e Tecidos Santo Antonio.
// Máquina: LINHA 1 DENIN - O.S.: 24.626
   VAR_TEMP
      AUX_R : Real;
   END_VAR
   VAR_TEMP   // added for the SCL form of the ladder/FBD networks
      _w1 : Bool;
   END_VAR
BEGIN

REGION Network 1: ALARMES
   // RESET DOS ALARMES
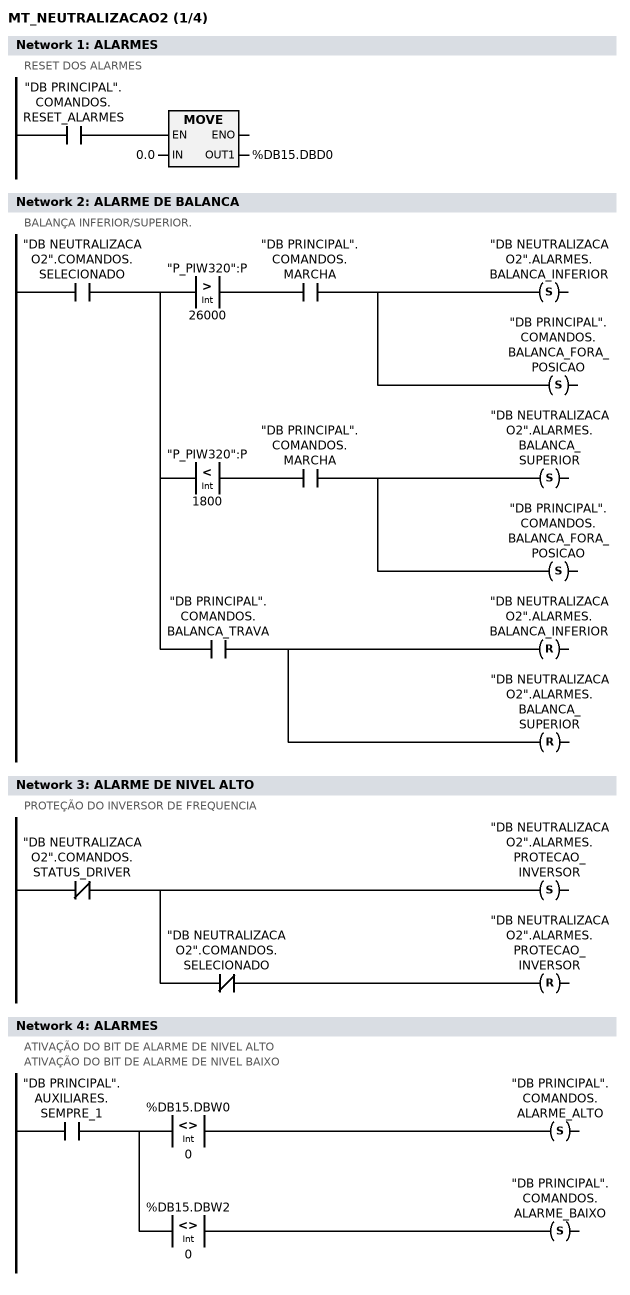
   RUNG wire#powerrail
      Contact( "DB PRINCIPAL".COMANDOS.RESET_ALARMES )
      { S7_GenerateENO := "TRUE" } Move(in := 0.0, out1 => %DB15.DBD0)
   END_RUNG
   // the same network as SCL:
   IF "DB PRINCIPAL".COMANDOS.RESET_ALARMES THEN %DB15.DBD0 := 0.0; END_IF;
END_REGION

REGION Network 2: ALARME DE BALANCA
   // BALANÇA INFERIOR/SUPERIOR.
   RUNG wire#powerrail
      Contact( "DB NEUTRALIZACAO2".COMANDOS.SELECIONADO )
      wire#w1
      { S7_Templates := "SrcType := Int" } GT_Contact(in1 := "P_PIW320":P, in2 := 26000)
      Contact( "DB PRINCIPAL".COMANDOS.MARCHA )
      wire#w2
      S_Coil( "DB NEUTRALIZACAO2".ALARMES.BALANCA_INFERIOR )
   END_RUNG
   RUNG wire#w2
      S_Coil( "DB PRINCIPAL".COMANDOS.BALANCA_FORA_POSICAO )
   END_RUNG
   RUNG wire#w1
      { S7_Templates := "SrcType := Int" } LT_Contact(in1 := "P_PIW320":P, in2 := 1800)
      Contact( "DB PRINCIPAL".COMANDOS.MARCHA )
      wire#w3
      S_Coil( "DB NEUTRALIZACAO2".ALARMES.BALANCA_SUPERIOR )
   END_RUNG
   RUNG wire#w3
      S_Coil( "DB PRINCIPAL".COMANDOS.BALANCA_FORA_POSICAO )
   END_RUNG
   RUNG wire#w1
      Contact( "DB PRINCIPAL".COMANDOS.BALANCA_TRAVA )
      wire#w4
      R_Coil( "DB NEUTRALIZACAO2".ALARMES.BALANCA_INFERIOR )
   END_RUNG
   RUNG wire#w4
      R_Coil( "DB NEUTRALIZACAO2".ALARMES.BALANCA_SUPERIOR )
   END_RUNG
   // the same network as SCL:
   IF "DB NEUTRALIZACAO2".COMANDOS.SELECIONADO AND ("P_PIW320":P > 26000) AND "DB PRINCIPAL".COMANDOS.MARCHA THEN
       "DB NEUTRALIZACAO2".ALARMES.BALANCA_INFERIOR := TRUE;
       "DB PRINCIPAL".COMANDOS.BALANCA_FORA_POSICAO := TRUE;
   END_IF;
   IF "DB NEUTRALIZACAO2".COMANDOS.SELECIONADO AND ("P_PIW320":P < 1800) AND "DB PRINCIPAL".COMANDOS.MARCHA THEN
       "DB NEUTRALIZACAO2".ALARMES.BALANCA_SUPERIOR := TRUE;
       "DB PRINCIPAL".COMANDOS.BALANCA_FORA_POSICAO := TRUE;
   END_IF;
   IF "DB NEUTRALIZACAO2".COMANDOS.SELECIONADO AND "DB PRINCIPAL".COMANDOS.BALANCA_TRAVA THEN
       "DB NEUTRALIZACAO2".ALARMES.BALANCA_INFERIOR := FALSE;
       "DB NEUTRALIZACAO2".ALARMES.BALANCA_SUPERIOR := FALSE;
   END_IF;
END_REGION

REGION Network 3: ALARME DE NIVEL ALTO
   // PROTEÇÃO DO INVERSOR DE FREQUENCIA
   RUNG wire#powerrail
      I_Contact( "DB NEUTRALIZACAO2".COMANDOS.STATUS_DRIVER )
      wire#w1
      S_Coil( "DB NEUTRALIZACAO2".ALARMES.PROTECAO_INVERSOR )
   END_RUNG
   RUNG wire#w1
      I_Contact( "DB NEUTRALIZACAO2".COMANDOS.SELECIONADO )
      R_Coil( "DB NEUTRALIZACAO2".ALARMES.PROTECAO_INVERSOR )
   END_RUNG
   // the same network as SCL:
   #_w1 := NOT "DB NEUTRALIZACAO2".COMANDOS.STATUS_DRIVER;
   IF #_w1 THEN "DB NEUTRALIZACAO2".ALARMES.PROTECAO_INVERSOR := TRUE; END_IF;
   IF #_w1 AND NOT "DB NEUTRALIZACAO2".COMANDOS.SELECIONADO THEN
       "DB NEUTRALIZACAO2".ALARMES.PROTECAO_INVERSOR := FALSE;
   END_IF;
END_REGION

REGION Network 4: ALARMES
   // ATIVAÇÃO DO BIT DE ALARME DE NIVEL ALTO
   // ATIVAÇÃO DO BIT DE ALARME DE NIVEL BAIXO
   RUNG wire#powerrail
      Contact( "DB PRINCIPAL".AUXILIARES.SEMPRE_1 )
      wire#w1
      { S7_Templates := "SrcType := Int" } NE_Contact(in1 := %DB15.DBW0, in2 := 0)
      S_Coil( "DB PRINCIPAL".COMANDOS.ALARME_ALTO )
   END_RUNG
   RUNG wire#w1
      { S7_Templates := "SrcType := Int" } NE_Contact(in1 := %DB15.DBW2, in2 := 0)
      S_Coil( "DB PRINCIPAL".COMANDOS.ALARME_BAIXO )
   END_RUNG
   // the same network as SCL:
   IF "DB PRINCIPAL".AUXILIARES.SEMPRE_1 AND (%DB15.DBW0 <> 0) THEN
       "DB PRINCIPAL".COMANDOS.ALARME_ALTO := TRUE;
   END_IF;
   IF "DB PRINCIPAL".AUXILIARES.SEMPRE_1 AND (%DB15.DBW2 <> 0) THEN
       "DB PRINCIPAL".COMANDOS.ALARME_BAIXO := TRUE;
   END_IF;
END_REGION

REGION Network 5: INDICAÇÃO DE MOTOR SELECIONADO
   // LIGA BIT QUE INDICA QUE HÁ ALGUM MOTOR SELECIONADO
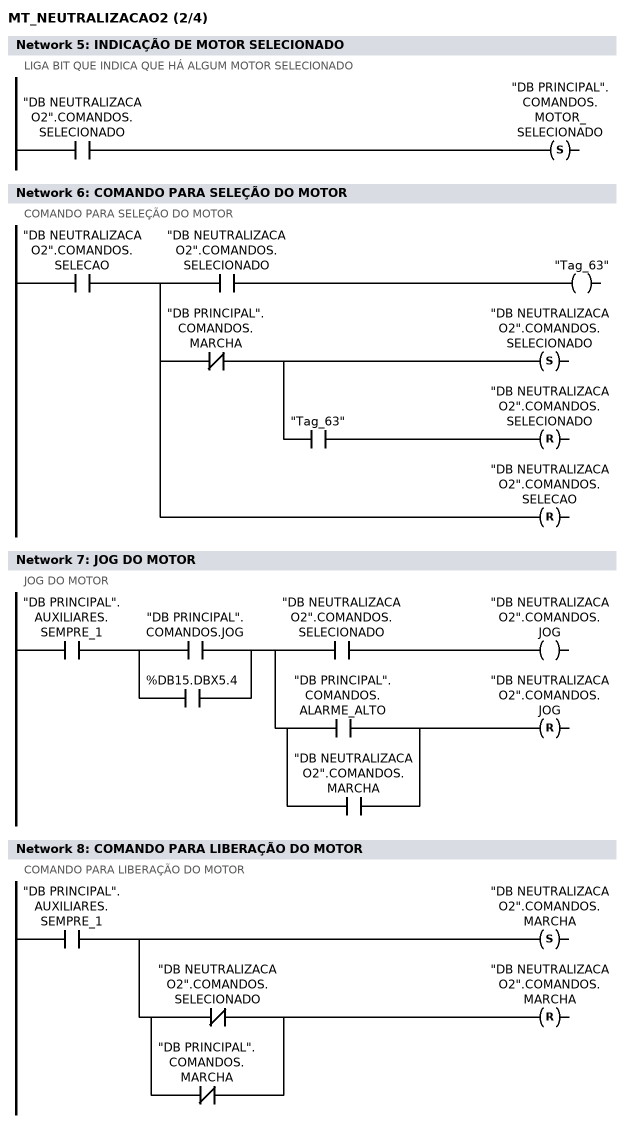
   RUNG wire#powerrail
      Contact( "DB NEUTRALIZACAO2".COMANDOS.SELECIONADO )
      S_Coil( "DB PRINCIPAL".COMANDOS.MOTOR_SELECIONADO )
   END_RUNG
   // the same network as SCL:
   IF "DB NEUTRALIZACAO2".COMANDOS.SELECIONADO THEN
       "DB PRINCIPAL".COMANDOS.MOTOR_SELECIONADO := TRUE;
   END_IF;
END_REGION

REGION Network 6: COMANDO PARA SELEÇÃO DO MOTOR
   // COMANDO PARA SELEÇÃO DO MOTOR
   RUNG wire#powerrail
      Contact( "DB NEUTRALIZACAO2".COMANDOS.SELECAO )
      wire#w1
      Contact( "DB NEUTRALIZACAO2".COMANDOS.SELECIONADO )
      Coil( "Tag_63" )
   END_RUNG
   RUNG wire#w1
      I_Contact( "DB PRINCIPAL".COMANDOS.MARCHA )
      wire#w2
      S_Coil( "DB NEUTRALIZACAO2".COMANDOS.SELECIONADO )
   END_RUNG
   RUNG wire#w2
      Contact( "Tag_63" )
      R_Coil( "DB NEUTRALIZACAO2".COMANDOS.SELECIONADO )
   END_RUNG
   RUNG wire#w1
      R_Coil( "DB NEUTRALIZACAO2".COMANDOS.SELECAO )
   END_RUNG
   // the same network as SCL:
   "Tag_63" := "DB NEUTRALIZACAO2".COMANDOS.SELECAO AND "DB NEUTRALIZACAO2".COMANDOS.SELECIONADO;
   #_w1 := "DB NEUTRALIZACAO2".COMANDOS.SELECAO AND NOT "DB PRINCIPAL".COMANDOS.MARCHA;
   IF #_w1 THEN "DB NEUTRALIZACAO2".COMANDOS.SELECIONADO := TRUE; END_IF;
   IF #_w1 AND "Tag_63" THEN "DB NEUTRALIZACAO2".COMANDOS.SELECIONADO := FALSE; END_IF;
   IF "DB NEUTRALIZACAO2".COMANDOS.SELECAO THEN "DB NEUTRALIZACAO2".COMANDOS.SELECAO := FALSE; END_IF;
END_REGION

REGION Network 7: JOG DO MOTOR
   // JOG DO MOTOR
   RUNG wire#powerrail
      Contact( "DB PRINCIPAL".AUXILIARES.SEMPRE_1 )
      wire#w1
      Contact( "DB PRINCIPAL".COMANDOS.JOG )
      wire#w2
      Contact( "DB NEUTRALIZACAO2".COMANDOS.SELECIONADO )
      Coil( "DB NEUTRALIZACAO2".COMANDOS.JOG )
   END_RUNG
   RUNG wire#w1
      Contact( %DB15.DBX5.4 )
   END_RUNG wire#w2
   RUNG wire#w2
      Contact( "DB PRINCIPAL".COMANDOS.ALARME_ALTO )
      wire#w3
      R_Coil( "DB NEUTRALIZACAO2".COMANDOS.JOG )
   END_RUNG
   RUNG wire#w2
      Contact( "DB NEUTRALIZACAO2".COMANDOS.MARCHA )
   END_RUNG wire#w3
   // the same network as SCL:
   #_w1 := "DB PRINCIPAL".AUXILIARES.SEMPRE_1 AND ("DB PRINCIPAL".COMANDOS.JOG OR %DB15.DBX5.4);
   "DB NEUTRALIZACAO2".COMANDOS.JOG := #_w1 AND "DB NEUTRALIZACAO2".COMANDOS.SELECIONADO;
   IF #_w1 AND ("DB PRINCIPAL".COMANDOS.ALARME_ALTO OR "DB NEUTRALIZACAO2".COMANDOS.MARCHA) THEN
       "DB NEUTRALIZACAO2".COMANDOS.JOG := FALSE;
   END_IF;
END_REGION

REGION Network 8: COMANDO PARA LIBERAÇÃO DO MOTOR
   // COMANDO PARA LIBERAÇÃO DO MOTOR
   RUNG wire#powerrail
      Contact( "DB PRINCIPAL".AUXILIARES.SEMPRE_1 )
      wire#w1
      S_Coil( "DB NEUTRALIZACAO2".COMANDOS.MARCHA )
   END_RUNG
   RUNG wire#w1
      I_Contact( "DB NEUTRALIZACAO2".COMANDOS.SELECIONADO )
      wire#w2
      R_Coil( "DB NEUTRALIZACAO2".COMANDOS.MARCHA )
   END_RUNG
   RUNG wire#w1
      I_Contact( "DB PRINCIPAL".COMANDOS.MARCHA )
   END_RUNG wire#w2
   // the same network as SCL:
   IF "DB PRINCIPAL".AUXILIARES.SEMPRE_1 THEN "DB NEUTRALIZACAO2".COMANDOS.MARCHA := TRUE; END_IF;
   IF "DB PRINCIPAL".AUXILIARES.SEMPRE_1 AND (NOT "DB NEUTRALIZACAO2".COMANDOS.SELECIONADO OR NOT "DB PRINCIPAL".COMANDOS.MARCHA) THEN
       "DB NEUTRALIZACAO2".COMANDOS.MARCHA := FALSE;
   END_IF;
END_REGION

REGION Network 9
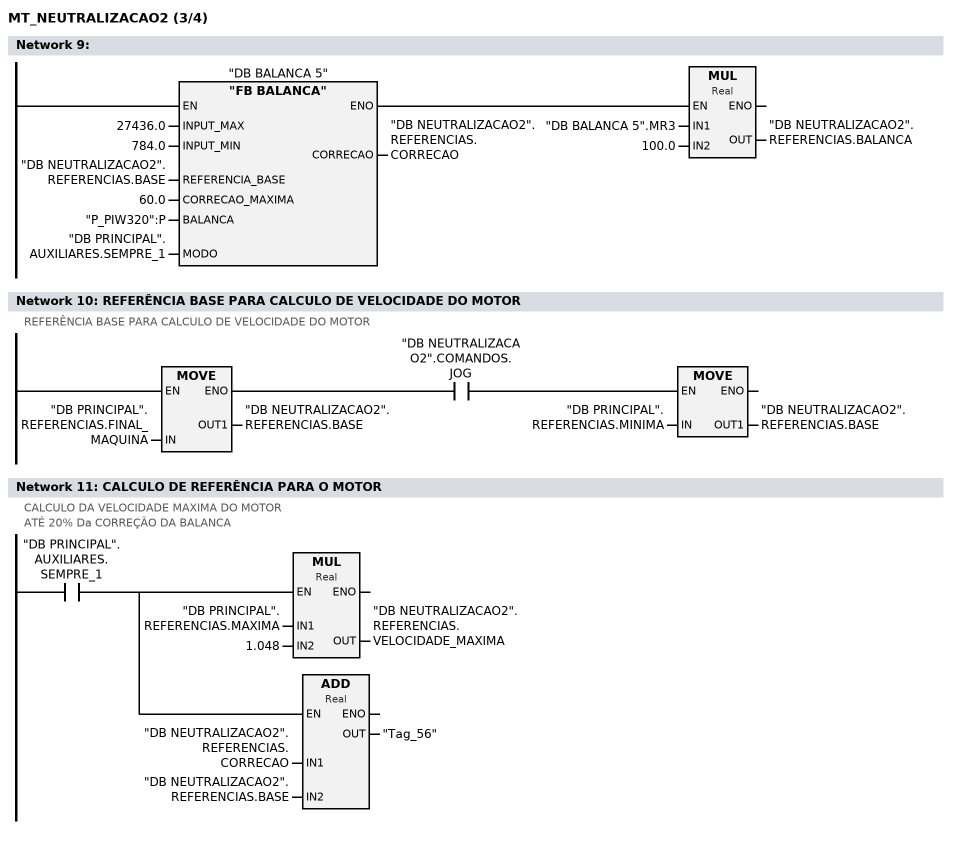
   RUNG wire#powerrail
      "DB BALANCA 5"(INPUT_MAX := 27436.0, INPUT_MIN := 784.0, REFERENCIA_BASE := "DB NEUTRALIZACAO2".REFERENCIAS.BASE, CORRECAO_MAXIMA := 60.0, BALANCA := "P_PIW320":P, MODO := "DB PRINCIPAL".AUXILIARES.SEMPRE_1, CORRECAO => "DB NEUTRALIZACAO2".REFERENCIAS.CORRECAO)
      { S7_Templates := "SrcType := Real"; S7_GenerateENO := "TRUE" } Mul(in1 := "DB BALANCA 5".MR3, in2 := 100.0, out => "DB NEUTRALIZACAO2".REFERENCIAS.BALANCA)
   END_RUNG
   // the same network as SCL:
   "DB BALANCA 5"(INPUT_MAX := 27436.0,   // "FB BALANCA"
                  INPUT_MIN := 784.0,
                  REFERENCIA_BASE := "DB NEUTRALIZACAO2".REFERENCIAS.BASE,
                  CORRECAO_MAXIMA := 60.0,
                  BALANCA := "P_PIW320":P,
                  MODO := "DB PRINCIPAL".AUXILIARES.SEMPRE_1,
                  CORRECAO => "DB NEUTRALIZACAO2".REFERENCIAS.CORRECAO,
                  ENO => #_w1);
   IF #_w1 THEN "DB NEUTRALIZACAO2".REFERENCIAS.BALANCA := "DB BALANCA 5".MR3 * 100.0; END_IF;
END_REGION

REGION Network 10: REFERÊNCIA BASE PARA CALCULO DE VELOCIDADE DO MOTOR
   // REFERÊNCIA BASE PARA CALCULO DE VELOCIDADE DO MOTOR
   RUNG wire#powerrail
      { S7_GenerateENO := "TRUE" } Move(in := "DB PRINCIPAL".REFERENCIAS.FINAL_MAQUINA, out1 => "DB NEUTRALIZACAO2".REFERENCIAS.BASE)
      Contact( "DB NEUTRALIZACAO2".COMANDOS.JOG )
      { S7_GenerateENO := "TRUE" } Move(in := "DB PRINCIPAL".REFERENCIAS.MINIMA, out1 => "DB NEUTRALIZACAO2".REFERENCIAS.BASE)
   END_RUNG
   // the same network as SCL:
   // ENO of a box is taken as its EN; it also drops when the box reports an error
   "DB NEUTRALIZACAO2".REFERENCIAS.BASE := "DB PRINCIPAL".REFERENCIAS.FINAL_MAQUINA;
   IF "DB NEUTRALIZACAO2".COMANDOS.JOG THEN
       "DB NEUTRALIZACAO2".REFERENCIAS.BASE := "DB PRINCIPAL".REFERENCIAS.MINIMA;
   END_IF;
END_REGION

REGION Network 11: CALCULO DE REFERÊNCIA PARA O MOTOR
   // CALCULO DA VELOCIDADE MAXIMA DO MOTOR
   // ATÉ 20% Da CORREÇÃO DA BALANCA
   RUNG wire#powerrail
      Contact( "DB PRINCIPAL".AUXILIARES.SEMPRE_1 )
      wire#w1
      { S7_Templates := "SrcType := Real"; S7_GenerateENO := "TRUE" } Mul(in1 := "DB PRINCIPAL".REFERENCIAS.MAXIMA, in2 := 1.048, out => "DB NEUTRALIZACAO2".REFERENCIAS.VELOCIDADE_MAXIMA)
   END_RUNG
   RUNG wire#w1
      { S7_Templates := "SrcType := Real"; S7_GenerateENO := "TRUE" } Add(in1 := "DB NEUTRALIZACAO2".REFERENCIAS.CORRECAO, in2 := "DB NEUTRALIZACAO2".REFERENCIAS.BASE, out => "Tag_56")
   END_RUNG
   // the same network as SCL:
   IF "DB PRINCIPAL".AUXILIARES.SEMPRE_1 THEN
       "DB NEUTRALIZACAO2".REFERENCIAS.VELOCIDADE_MAXIMA := "DB PRINCIPAL".REFERENCIAS.MAXIMA * 1.048;
       "Tag_56" := "DB NEUTRALIZACAO2".REFERENCIAS.CORRECAO + "DB NEUTRALIZACAO2".REFERENCIAS.BASE;
   END_IF;
END_REGION

REGION Network 12: ACC/DEC DA REFERÊNCIA DO MOTOR
   // ACC/DEC DA REFERÊNCIA DO MOTOR
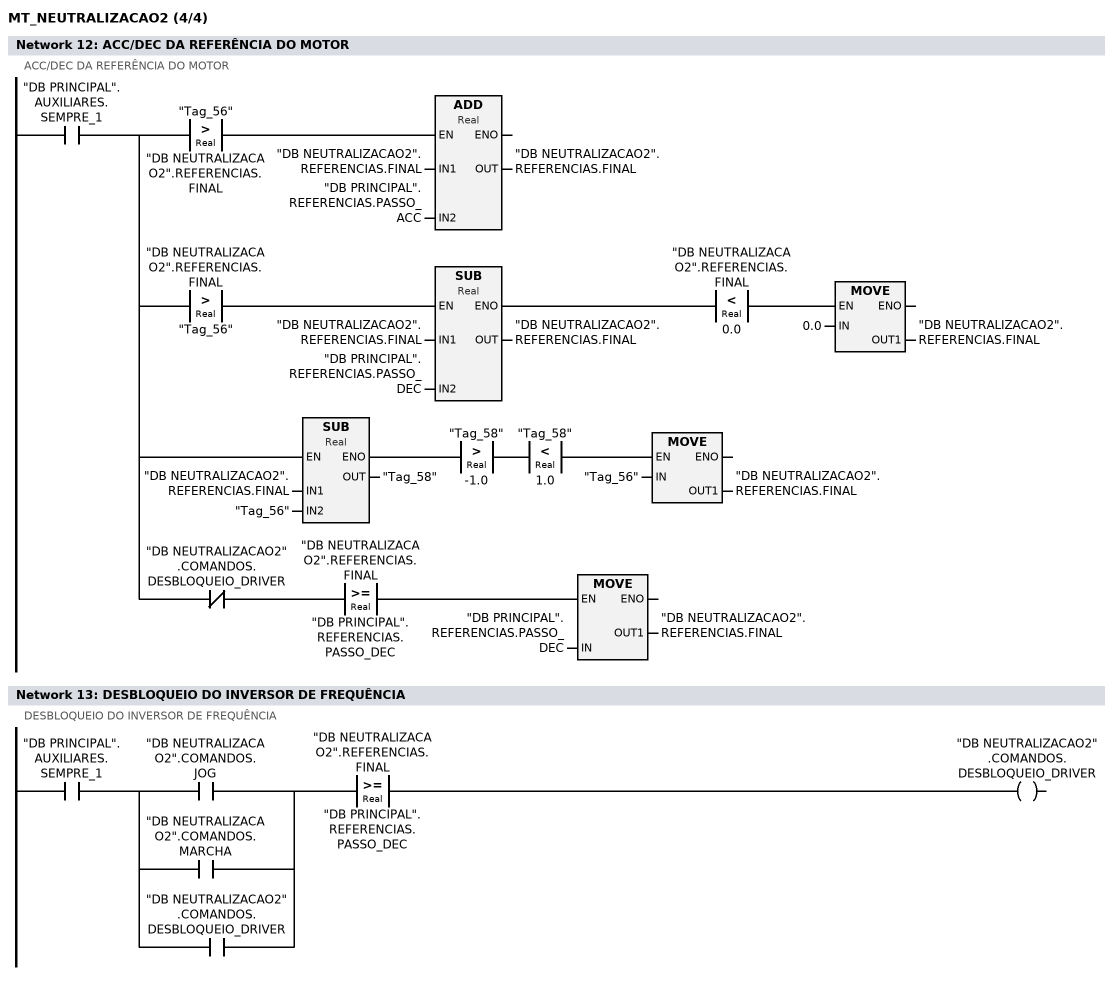
   RUNG wire#powerrail
      Contact( "DB PRINCIPAL".AUXILIARES.SEMPRE_1 )
      wire#w1
      { S7_Templates := "SrcType := Real" } GT_Contact(in1 := "Tag_56", in2 := "DB NEUTRALIZACAO2".REFERENCIAS.FINAL)
      { S7_Templates := "SrcType := Real"; S7_GenerateENO := "TRUE" } Add(in1 := "DB NEUTRALIZACAO2".REFERENCIAS.FINAL, in2 := "DB PRINCIPAL".REFERENCIAS.PASSO_ACC, out => "DB NEUTRALIZACAO2".REFERENCIAS.FINAL)
   END_RUNG
   RUNG wire#w1
      { S7_Templates := "SrcType := Real" } GT_Contact(in1 := "DB NEUTRALIZACAO2".REFERENCIAS.FINAL, in2 := "Tag_56")
      { S7_Templates := "SrcType := Real"; S7_GenerateENO := "TRUE" } Sub(in1 := "DB NEUTRALIZACAO2".REFERENCIAS.FINAL, in2 := "DB PRINCIPAL".REFERENCIAS.PASSO_DEC, out => "DB NEUTRALIZACAO2".REFERENCIAS.FINAL)
      { S7_Templates := "SrcType := Real" } LT_Contact(in1 := "DB NEUTRALIZACAO2".REFERENCIAS.FINAL, in2 := 0.0)
      { S7_GenerateENO := "TRUE" } Move(in := 0.0, out1 => "DB NEUTRALIZACAO2".REFERENCIAS.FINAL)
   END_RUNG
   RUNG wire#w1
      { S7_Templates := "SrcType := Real"; S7_GenerateENO := "TRUE" } Sub(in1 := "DB NEUTRALIZACAO2".REFERENCIAS.FINAL, in2 := "Tag_56", out => "Tag_58")
      { S7_Templates := "SrcType := Real" } GT_Contact(in1 := "Tag_58", in2 := -1.0)
      { S7_Templates := "SrcType := Real" } LT_Contact(in1 := "Tag_58", in2 := 1.0)
      { S7_GenerateENO := "TRUE" } Move(in := "Tag_56", out1 => "DB NEUTRALIZACAO2".REFERENCIAS.FINAL)
   END_RUNG
   RUNG wire#w1
      I_Contact( "DB NEUTRALIZACAO2".COMANDOS.DESBLOQUEIO_DRIVER )
      { S7_Templates := "SrcType := Real" } GE_Contact(in1 := "DB NEUTRALIZACAO2".REFERENCIAS.FINAL, in2 := "DB PRINCIPAL".REFERENCIAS.PASSO_DEC)
      { S7_GenerateENO := "TRUE" } Move(in := "DB PRINCIPAL".REFERENCIAS.PASSO_DEC, out1 => "DB NEUTRALIZACAO2".REFERENCIAS.FINAL)
   END_RUNG
   // the same network as SCL:
   // ENO of a box is taken as its EN; it also drops when the box reports an error
   IF "DB PRINCIPAL".AUXILIARES.SEMPRE_1 AND ("Tag_56" > "DB NEUTRALIZACAO2".REFERENCIAS.FINAL) THEN
       "DB NEUTRALIZACAO2".REFERENCIAS.FINAL := "DB NEUTRALIZACAO2".REFERENCIAS.FINAL + "DB PRINCIPAL".REFERENCIAS.PASSO_ACC;
   END_IF;
   #_w1 := "DB PRINCIPAL".AUXILIARES.SEMPRE_1 AND ("DB NEUTRALIZACAO2".REFERENCIAS.FINAL > "Tag_56");
   IF #_w1 THEN
       "DB NEUTRALIZACAO2".REFERENCIAS.FINAL := "DB NEUTRALIZACAO2".REFERENCIAS.FINAL - "DB PRINCIPAL".REFERENCIAS.PASSO_DEC;
   END_IF;
   IF #_w1 AND ("DB NEUTRALIZACAO2".REFERENCIAS.FINAL < 0.0) THEN
       "DB NEUTRALIZACAO2".REFERENCIAS.FINAL := 0.0;
   END_IF;
   IF "DB PRINCIPAL".AUXILIARES.SEMPRE_1 THEN
       "Tag_58" := "DB NEUTRALIZACAO2".REFERENCIAS.FINAL - "Tag_56";
   END_IF;
   IF "DB PRINCIPAL".AUXILIARES.SEMPRE_1 AND ("Tag_58" > (-1.0)) AND ("Tag_58" < 1.0) THEN
       "DB NEUTRALIZACAO2".REFERENCIAS.FINAL := "Tag_56";
   END_IF;
   IF "DB PRINCIPAL".AUXILIARES.SEMPRE_1 AND NOT "DB NEUTRALIZACAO2".COMANDOS.DESBLOQUEIO_DRIVER AND ("DB NEUTRALIZACAO2".REFERENCIAS.FINAL >= "DB PRINCIPAL".REFERENCIAS.PASSO_DEC) THEN
       "DB NEUTRALIZACAO2".REFERENCIAS.FINAL := "DB PRINCIPAL".REFERENCIAS.PASSO_DEC;
   END_IF;
END_REGION

REGION Network 13: DESBLOQUEIO DO INVERSOR DE FREQUÊNCIA
   // DESBLOQUEIO DO INVERSOR DE FREQUÊNCIA
   RUNG wire#powerrail
      Contact( "DB PRINCIPAL".AUXILIARES.SEMPRE_1 )
      wire#w1
      Contact( "DB NEUTRALIZACAO2".COMANDOS.JOG )
      wire#w2
      { S7_Templates := "SrcType := Real" } GE_Contact(in1 := "DB NEUTRALIZACAO2".REFERENCIAS.FINAL, in2 := "DB PRINCIPAL".REFERENCIAS.PASSO_DEC)
      Coil( "DB NEUTRALIZACAO2".COMANDOS.DESBLOQUEIO_DRIVER )
   END_RUNG
   RUNG wire#w1
      Contact( "DB NEUTRALIZACAO2".COMANDOS.MARCHA )
   END_RUNG wire#w2
   RUNG wire#w1
      Contact( "DB NEUTRALIZACAO2".COMANDOS.DESBLOQUEIO_DRIVER )
   END_RUNG wire#w2
   // the same network as SCL:
   "DB NEUTRALIZACAO2".COMANDOS.DESBLOQUEIO_DRIVER := "DB PRINCIPAL".AUXILIARES.SEMPRE_1 AND ("DB NEUTRALIZACAO2".COMANDOS.JOG OR "DB NEUTRALIZACAO2".COMANDOS.MARCHA OR "DB NEUTRALIZACAO2".COMANDOS.DESBLOQUEIO_DRIVER) AND ("DB NEUTRALIZACAO2".REFERENCIAS.FINAL >= "DB PRINCIPAL".REFERENCIAS.PASSO_DEC);
END_REGION

REGION Network 14: STATUS / CONTROLE - INVERSOR DE FREQUÊNCIA
   // DANFOSS FC300 PROFIBUS - TEX24626INV001
END_REGION

REGION Network 15 (STL): INVERSOR RESERVA
         A     "DB PRINCIPAL".AUXILIARES.SEMPRE_1;
         =     %L24.0;
         A     %L24.0;
         A(;
         L     "DB PRINCIPAL".AUXILIARES1.INVERSOR_RESERVA1;
         L     6;
         ==I;
         );
         =     %L24.1;
         A     %L24.1;
         JNB   M001;
         L     "DB NEUTRALIZACAO2".REFERENCIAS.FINAL;
         L     3.456;
         *R;
         T     #AUX_R;
         RND;
         T     "P_QW100":P;
   M001: NOP   0;
         A     %L24.1;
         A     "I130";
         S     "DB PRINCIPAL".ALARME.INV_RESERVA1;
         A     %L24.1;
         A     "DB NEUTRALIZACAO2".COMANDOS.DESBLOQUEIO_DRIVER;
         S     "Q134";
         A     %L24.1;
         AN    "DB NEUTRALIZACAO2".COMANDOS.DESBLOQUEIO_DRIVER;
         R     "Q134";
         A     %L24.0;
         A(;
         L     "DB PRINCIPAL".AUXILIARES1.INVERSOR_RESERVA2;
         L     6;
         ==I;
         );
         =     %L24.1;
         A     %L24.1;
         JNB   M002;
         L     "DB NEUTRALIZACAO2".REFERENCIAS.FINAL;
         L     3.456;
         *R;
         T     #AUX_R;
         RND;
         T     "P_QW102":P;
   M002: NOP   0;
         A     %L24.1;
         A     "I132";
         S     "DB PRINCIPAL".ALARME.INV_RESERVA2;
         A     %L24.1;
         A     "DB NEUTRALIZACAO2".COMANDOS.DESBLOQUEIO_DRIVER;
         S     "Q135";
         A     %L24.1;
         AN    "DB NEUTRALIZACAO2".COMANDOS.DESBLOQUEIO_DRIVER;
         R     "Q135";
END_REGION
END_FUNCTION

FUNCTION "MT_EXTRACTA2" : Void   // FC16, LAD
TITLE = MÓDULO DE CONTROLE DA EXTRACTA 2
{ S7_Optimized_Access := 'FALSE' }
AUTHOR : THALLES
FAMILY : TRAÇÃO
NAME : LINHA1
VERSION : 0.1
// DATA BLOCK DE CONTROLE // DB16
// Automation Pack Automação Indl. e Com. Ltda.
// Cliente: Texima S/A Ind. de Máquinas
// Cliente Final: Cia. Fiação e Tecidos Santo Antonio.
// Máquina: LINHA 1 DENIN - O.S.: 24.626
   VAR_TEMP
      AUX_R : Real;
   END_VAR
   VAR_TEMP   // added for the SCL form of the ladder/FBD networks
      _w1 : Bool;
      _w2 : Bool;
   END_VAR
BEGIN

REGION Network 1: ALARMES
   // RESET DOS ALARMES
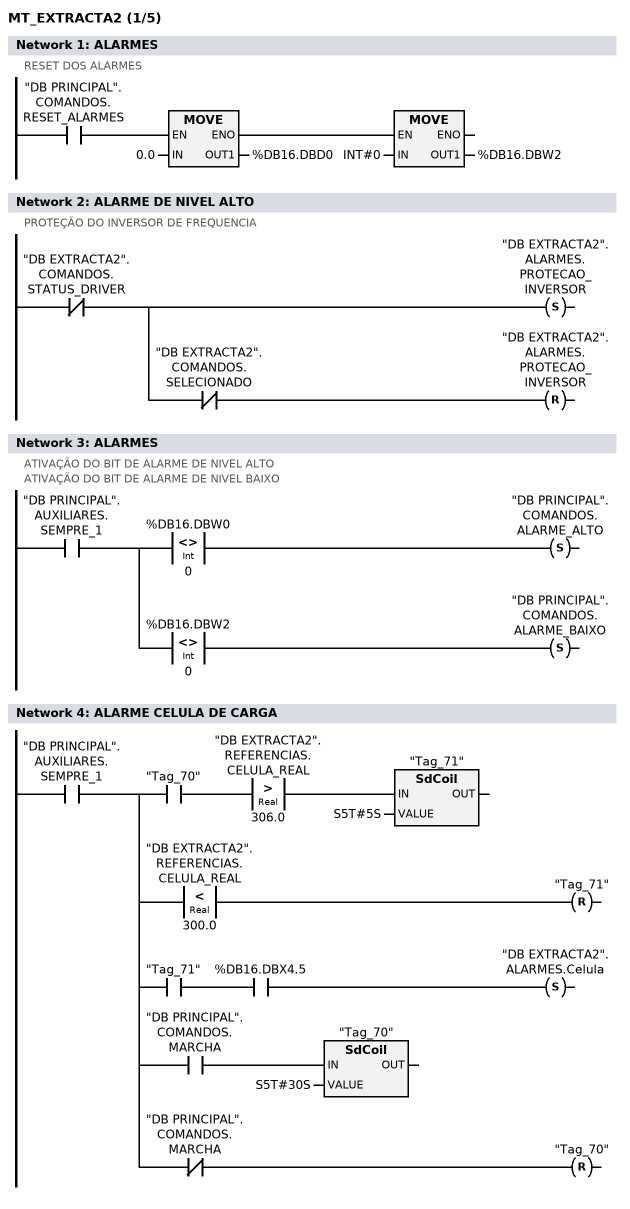
   RUNG wire#powerrail
      Contact( "DB PRINCIPAL".COMANDOS.RESET_ALARMES )
      { S7_GenerateENO := "TRUE" } Move(in := 0.0, out1 => %DB16.DBD0)
      { S7_GenerateENO := "TRUE" } Move(in := INT#0, out1 => %DB16.DBW2)
   END_RUNG
   // the same network as SCL:
   // ENO of a box is taken as its EN; it also drops when the box reports an error
   IF "DB PRINCIPAL".COMANDOS.RESET_ALARMES THEN
       %DB16.DBD0 := 0.0;
       %DB16.DBW2 := INT#0;
   END_IF;
END_REGION

REGION Network 2: ALARME DE NIVEL ALTO
   // PROTEÇÃO DO INVERSOR DE FREQUENCIA
   RUNG wire#powerrail
      I_Contact( "DB EXTRACTA2".COMANDOS.STATUS_DRIVER )
      wire#w1
      S_Coil( "DB EXTRACTA2".ALARMES.PROTECAO_INVERSOR )
   END_RUNG
   RUNG wire#w1
      I_Contact( "DB EXTRACTA2".COMANDOS.SELECIONADO )
      R_Coil( "DB EXTRACTA2".ALARMES.PROTECAO_INVERSOR )
   END_RUNG
   // the same network as SCL:
   #_w1 := NOT "DB EXTRACTA2".COMANDOS.STATUS_DRIVER;
   IF #_w1 THEN "DB EXTRACTA2".ALARMES.PROTECAO_INVERSOR := TRUE; END_IF;
   IF #_w1 AND NOT "DB EXTRACTA2".COMANDOS.SELECIONADO THEN
       "DB EXTRACTA2".ALARMES.PROTECAO_INVERSOR := FALSE;
   END_IF;
END_REGION

REGION Network 3: ALARMES
   // ATIVAÇÃO DO BIT DE ALARME DE NIVEL ALTO
   // ATIVAÇÃO DO BIT DE ALARME DE NIVEL BAIXO
   RUNG wire#powerrail
      Contact( "DB PRINCIPAL".AUXILIARES.SEMPRE_1 )
      wire#w1
      { S7_Templates := "SrcType := Int" } NE_Contact(in1 := %DB16.DBW0, in2 := 0)
      S_Coil( "DB PRINCIPAL".COMANDOS.ALARME_ALTO )
   END_RUNG
   RUNG wire#w1
      { S7_Templates := "SrcType := Int" } NE_Contact(in1 := %DB16.DBW2, in2 := 0)
      S_Coil( "DB PRINCIPAL".COMANDOS.ALARME_BAIXO )
   END_RUNG
   // the same network as SCL:
   IF "DB PRINCIPAL".AUXILIARES.SEMPRE_1 AND (%DB16.DBW0 <> 0) THEN
       "DB PRINCIPAL".COMANDOS.ALARME_ALTO := TRUE;
   END_IF;
   IF "DB PRINCIPAL".AUXILIARES.SEMPRE_1 AND (%DB16.DBW2 <> 0) THEN
       "DB PRINCIPAL".COMANDOS.ALARME_BAIXO := TRUE;
   END_IF;
END_REGION

REGION Network 4: ALARME CELULA DE CARGA
   // no SCL statement known for SdCoil: written as a call
   #_w1 := "DB PRINCIPAL".AUXILIARES.SEMPRE_1;
   SdCoil(value := S5T#5S,
          in := "DB PRINCIPAL".AUXILIARES.SEMPRE_1 AND "Tag_70" AND ("DB EXTRACTA2".REFERENCIAS.CELULA_REAL > 306.0),
          operand := "Tag_71");
   IF #_w1 AND ("DB EXTRACTA2".REFERENCIAS.CELULA_REAL < 300.0) THEN "Tag_71" := FALSE; END_IF;
   IF #_w1 AND "Tag_71" AND %DB16.DBX4.5 THEN "DB EXTRACTA2".ALARMES.Celula := TRUE; END_IF;
   SdCoil(value := S5T#30S, operand := "Tag_70", in := #_w1 AND "DB PRINCIPAL".COMANDOS.MARCHA);
   IF #_w1 AND NOT "DB PRINCIPAL".COMANDOS.MARCHA THEN "Tag_70" := FALSE; END_IF;
END_REGION

REGION Network 5: INDICAÇÃO DE MOTOR SELECIONADO
   // LIGA BIT QUE INDICA QUE HÁ ALGUM MOTOR SELECIONADO
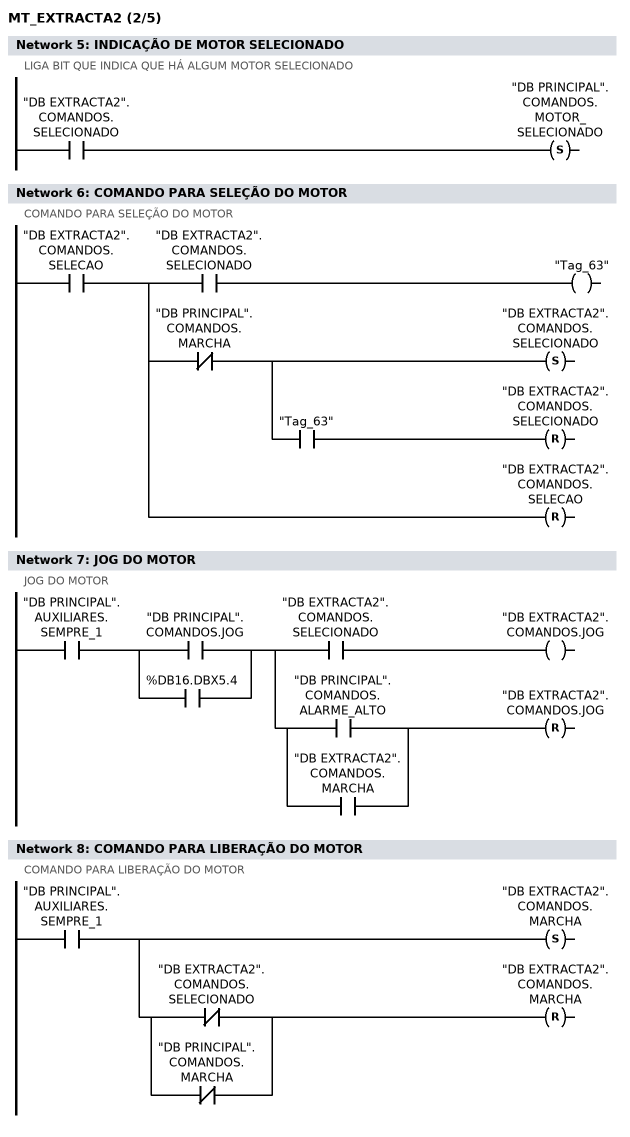
   RUNG wire#powerrail
      Contact( "DB EXTRACTA2".COMANDOS.SELECIONADO )
      S_Coil( "DB PRINCIPAL".COMANDOS.MOTOR_SELECIONADO )
   END_RUNG
   // the same network as SCL:
   IF "DB EXTRACTA2".COMANDOS.SELECIONADO THEN "DB PRINCIPAL".COMANDOS.MOTOR_SELECIONADO := TRUE; END_IF;
END_REGION

REGION Network 6: COMANDO PARA SELEÇÃO DO MOTOR
   // COMANDO PARA SELEÇÃO DO MOTOR
   RUNG wire#powerrail
      Contact( "DB EXTRACTA2".COMANDOS.SELECAO )
      wire#w1
      Contact( "DB EXTRACTA2".COMANDOS.SELECIONADO )
      Coil( "Tag_63" )
   END_RUNG
   RUNG wire#w1
      I_Contact( "DB PRINCIPAL".COMANDOS.MARCHA )
      wire#w2
      S_Coil( "DB EXTRACTA2".COMANDOS.SELECIONADO )
   END_RUNG
   RUNG wire#w2
      Contact( "Tag_63" )
      R_Coil( "DB EXTRACTA2".COMANDOS.SELECIONADO )
   END_RUNG
   RUNG wire#w1
      R_Coil( "DB EXTRACTA2".COMANDOS.SELECAO )
   END_RUNG
   // the same network as SCL:
   "Tag_63" := "DB EXTRACTA2".COMANDOS.SELECAO AND "DB EXTRACTA2".COMANDOS.SELECIONADO;
   #_w1 := "DB EXTRACTA2".COMANDOS.SELECAO AND NOT "DB PRINCIPAL".COMANDOS.MARCHA;
   IF #_w1 THEN "DB EXTRACTA2".COMANDOS.SELECIONADO := TRUE; END_IF;
   IF #_w1 AND "Tag_63" THEN "DB EXTRACTA2".COMANDOS.SELECIONADO := FALSE; END_IF;
   IF "DB EXTRACTA2".COMANDOS.SELECAO THEN "DB EXTRACTA2".COMANDOS.SELECAO := FALSE; END_IF;
END_REGION

REGION Network 7: JOG DO MOTOR
   // JOG DO MOTOR
   RUNG wire#powerrail
      Contact( "DB PRINCIPAL".AUXILIARES.SEMPRE_1 )
      wire#w1
      Contact( "DB PRINCIPAL".COMANDOS.JOG )
      wire#w2
      Contact( "DB EXTRACTA2".COMANDOS.SELECIONADO )
      Coil( "DB EXTRACTA2".COMANDOS.JOG )
   END_RUNG
   RUNG wire#w1
      Contact( %DB16.DBX5.4 )
   END_RUNG wire#w2
   RUNG wire#w2
      Contact( "DB PRINCIPAL".COMANDOS.ALARME_ALTO )
      wire#w3
      R_Coil( "DB EXTRACTA2".COMANDOS.JOG )
   END_RUNG
   RUNG wire#w2
      Contact( "DB EXTRACTA2".COMANDOS.MARCHA )
   END_RUNG wire#w3
   // the same network as SCL:
   #_w1 := "DB PRINCIPAL".AUXILIARES.SEMPRE_1 AND ("DB PRINCIPAL".COMANDOS.JOG OR %DB16.DBX5.4);
   "DB EXTRACTA2".COMANDOS.JOG := #_w1 AND "DB EXTRACTA2".COMANDOS.SELECIONADO;
   IF #_w1 AND ("DB PRINCIPAL".COMANDOS.ALARME_ALTO OR "DB EXTRACTA2".COMANDOS.MARCHA) THEN
       "DB EXTRACTA2".COMANDOS.JOG := FALSE;
   END_IF;
END_REGION

REGION Network 8: COMANDO PARA LIBERAÇÃO DO MOTOR
   // COMANDO PARA LIBERAÇÃO DO MOTOR
   RUNG wire#powerrail
      Contact( "DB PRINCIPAL".AUXILIARES.SEMPRE_1 )
      wire#w1
      S_Coil( "DB EXTRACTA2".COMANDOS.MARCHA )
   END_RUNG
   RUNG wire#w1
      I_Contact( "DB EXTRACTA2".COMANDOS.SELECIONADO )
      wire#w2
      R_Coil( "DB EXTRACTA2".COMANDOS.MARCHA )
   END_RUNG
   RUNG wire#w1
      I_Contact( "DB PRINCIPAL".COMANDOS.MARCHA )
   END_RUNG wire#w2
   // the same network as SCL:
   IF "DB PRINCIPAL".AUXILIARES.SEMPRE_1 THEN "DB EXTRACTA2".COMANDOS.MARCHA := TRUE; END_IF;
   IF "DB PRINCIPAL".AUXILIARES.SEMPRE_1 AND (NOT "DB EXTRACTA2".COMANDOS.SELECIONADO OR NOT "DB PRINCIPAL".COMANDOS.MARCHA) THEN
       "DB EXTRACTA2".COMANDOS.MARCHA := FALSE;
   END_IF;
END_REGION

REGION Network 9: REFERÊNCIA BASE PARA CALCULO DE VELOCIDADE DO MOTOR
   // REFERÊNCIA BASE PARA CALCULO DE VELOCIDADE DO MOTOR
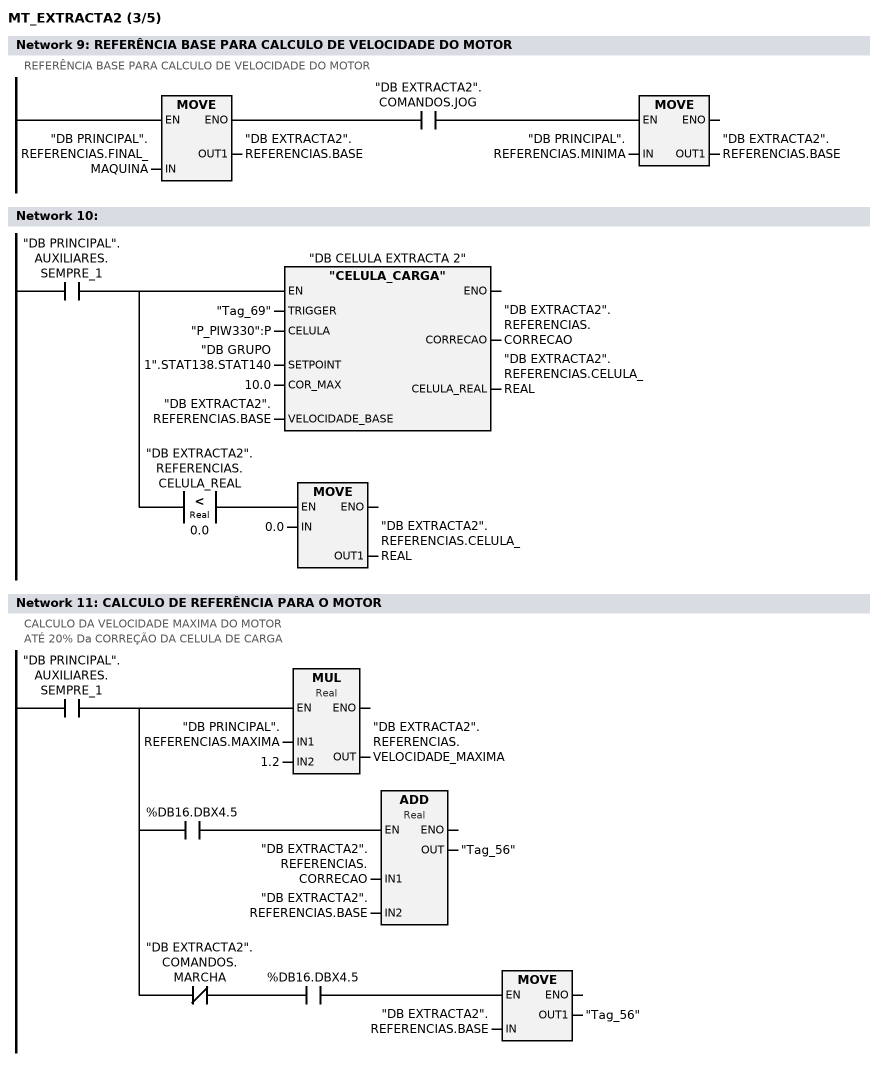
   RUNG wire#powerrail
      { S7_GenerateENO := "TRUE" } Move(in := "DB PRINCIPAL".REFERENCIAS.FINAL_MAQUINA, out1 => "DB EXTRACTA2".REFERENCIAS.BASE)
      Contact( "DB EXTRACTA2".COMANDOS.JOG )
      { S7_GenerateENO := "TRUE" } Move(in := "DB PRINCIPAL".REFERENCIAS.MINIMA, out1 => "DB EXTRACTA2".REFERENCIAS.BASE)
   END_RUNG
   // the same network as SCL:
   // ENO of a box is taken as its EN; it also drops when the box reports an error
   "DB EXTRACTA2".REFERENCIAS.BASE := "DB PRINCIPAL".REFERENCIAS.FINAL_MAQUINA;
   IF "DB EXTRACTA2".COMANDOS.JOG THEN
       "DB EXTRACTA2".REFERENCIAS.BASE := "DB PRINCIPAL".REFERENCIAS.MINIMA;
   END_IF;
END_REGION

REGION Network 10
   RUNG wire#powerrail
      Contact( "DB PRINCIPAL".AUXILIARES.SEMPRE_1 )
      wire#w1
      "DB CELULA EXTRACTA 2"(TRIGGER := "Tag_69", CELULA := "P_PIW330":P, SETPOINT := "DB GRUPO 1".STAT138.STAT140, COR_MAX := 10.0, VELOCIDADE_BASE := "DB EXTRACTA2".REFERENCIAS.BASE, CORRECAO => "DB EXTRACTA2".REFERENCIAS.CORRECAO, CELULA_REAL => "DB EXTRACTA2".REFERENCIAS.CELULA_REAL)
   END_RUNG
   RUNG wire#w1
      { S7_Templates := "SrcType := Real" } LT_Contact(in1 := "DB EXTRACTA2".REFERENCIAS.CELULA_REAL, in2 := 0.0)
      { S7_GenerateENO := "TRUE" } Move(in := 0.0, out1 => "DB EXTRACTA2".REFERENCIAS.CELULA_REAL)
   END_RUNG
   // the same network as SCL:
   #_w1 := "DB PRINCIPAL".AUXILIARES.SEMPRE_1;
   IF #_w1 THEN
       "DB CELULA EXTRACTA 2"(TRIGGER := "Tag_69",   // "CELULA_CARGA"
                              CELULA := "P_PIW330":P,
                              SETPOINT := "DB GRUPO 1".STAT138.STAT140,
                              COR_MAX := 10.0,
                              VELOCIDADE_BASE := "DB EXTRACTA2".REFERENCIAS.BASE,
                              CORRECAO => "DB EXTRACTA2".REFERENCIAS.CORRECAO,
                              CELULA_REAL => "DB EXTRACTA2".REFERENCIAS.CELULA_REAL);
   END_IF;
   IF #_w1 AND ("DB EXTRACTA2".REFERENCIAS.CELULA_REAL < 0.0) THEN
       "DB EXTRACTA2".REFERENCIAS.CELULA_REAL := 0.0;
   END_IF;
END_REGION

REGION Network 11: CALCULO DE REFERÊNCIA PARA O MOTOR
   // CALCULO DA VELOCIDADE MAXIMA DO MOTOR
   // ATÉ 20% Da CORREÇÃO DA CELULA DE CARGA
   RUNG wire#powerrail
      Contact( "DB PRINCIPAL".AUXILIARES.SEMPRE_1 )
      wire#w1
      { S7_Templates := "SrcType := Real"; S7_GenerateENO := "TRUE" } Mul(in1 := "DB PRINCIPAL".REFERENCIAS.MAXIMA, in2 := 1.2, out => "DB EXTRACTA2".REFERENCIAS.VELOCIDADE_MAXIMA)
   END_RUNG
   RUNG wire#w1
      Contact( %DB16.DBX4.5 )
      { S7_Templates := "SrcType := Real"; S7_GenerateENO := "TRUE" } Add(in1 := "DB EXTRACTA2".REFERENCIAS.CORRECAO, in2 := "DB EXTRACTA2".REFERENCIAS.BASE, out => "Tag_56")
   END_RUNG
   RUNG wire#w1
      I_Contact( "DB EXTRACTA2".COMANDOS.MARCHA )
      Contact( %DB16.DBX4.5 )
      { S7_GenerateENO := "TRUE" } Move(in := "DB EXTRACTA2".REFERENCIAS.BASE, out1 => "Tag_56")
   END_RUNG
   // the same network as SCL:
   IF "DB PRINCIPAL".AUXILIARES.SEMPRE_1 THEN
       "DB EXTRACTA2".REFERENCIAS.VELOCIDADE_MAXIMA := "DB PRINCIPAL".REFERENCIAS.MAXIMA * 1.2;
   END_IF;
   IF "DB PRINCIPAL".AUXILIARES.SEMPRE_1 AND %DB16.DBX4.5 THEN
       "Tag_56" := "DB EXTRACTA2".REFERENCIAS.CORRECAO + "DB EXTRACTA2".REFERENCIAS.BASE;
   END_IF;
   IF "DB PRINCIPAL".AUXILIARES.SEMPRE_1 AND NOT "DB EXTRACTA2".COMANDOS.MARCHA AND %DB16.DBX4.5 THEN
       "Tag_56" := "DB EXTRACTA2".REFERENCIAS.BASE;
   END_IF;
END_REGION

REGION Network 12: ACC/DEC DA REFERÊNCIA DO MOTOR
   // ACC/DEC DA REFERÊNCIA DO MOTOR
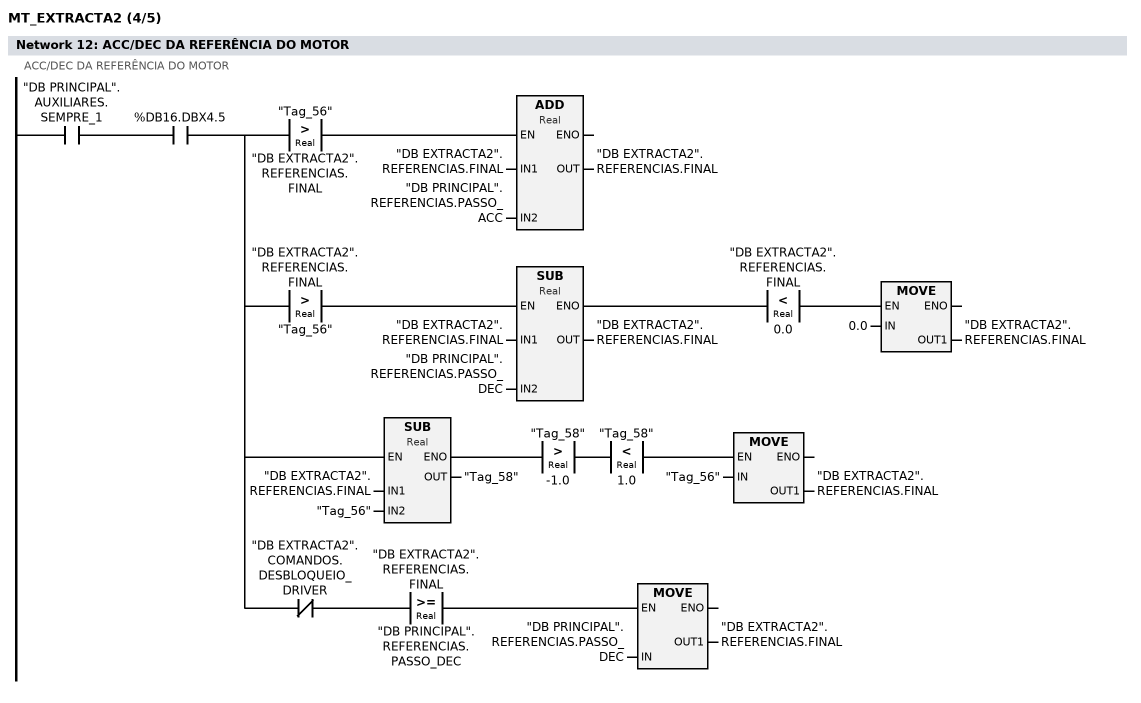
   RUNG wire#powerrail
      Contact( "DB PRINCIPAL".AUXILIARES.SEMPRE_1 )
      Contact( %DB16.DBX4.5 )
      wire#w1
      { S7_Templates := "SrcType := Real" } GT_Contact(in1 := "Tag_56", in2 := "DB EXTRACTA2".REFERENCIAS.FINAL)
      { S7_Templates := "SrcType := Real"; S7_GenerateENO := "TRUE" } Add(in1 := "DB EXTRACTA2".REFERENCIAS.FINAL, in2 := "DB PRINCIPAL".REFERENCIAS.PASSO_ACC, out => "DB EXTRACTA2".REFERENCIAS.FINAL)
   END_RUNG
   RUNG wire#w1
      { S7_Templates := "SrcType := Real" } GT_Contact(in1 := "DB EXTRACTA2".REFERENCIAS.FINAL, in2 := "Tag_56")
      { S7_Templates := "SrcType := Real"; S7_GenerateENO := "TRUE" } Sub(in1 := "DB EXTRACTA2".REFERENCIAS.FINAL, in2 := "DB PRINCIPAL".REFERENCIAS.PASSO_DEC, out => "DB EXTRACTA2".REFERENCIAS.FINAL)
      { S7_Templates := "SrcType := Real" } LT_Contact(in1 := "DB EXTRACTA2".REFERENCIAS.FINAL, in2 := 0.0)
      { S7_GenerateENO := "TRUE" } Move(in := 0.0, out1 => "DB EXTRACTA2".REFERENCIAS.FINAL)
   END_RUNG
   RUNG wire#w1
      { S7_Templates := "SrcType := Real"; S7_GenerateENO := "TRUE" } Sub(in1 := "DB EXTRACTA2".REFERENCIAS.FINAL, in2 := "Tag_56", out => "Tag_58")
      { S7_Templates := "SrcType := Real" } GT_Contact(in1 := "Tag_58", in2 := -1.0)
      { S7_Templates := "SrcType := Real" } LT_Contact(in1 := "Tag_58", in2 := 1.0)
      { S7_GenerateENO := "TRUE" } Move(in := "Tag_56", out1 => "DB EXTRACTA2".REFERENCIAS.FINAL)
   END_RUNG
   RUNG wire#w1
      I_Contact( "DB EXTRACTA2".COMANDOS.DESBLOQUEIO_DRIVER )
      { S7_Templates := "SrcType := Real" } GE_Contact(in1 := "DB EXTRACTA2".REFERENCIAS.FINAL, in2 := "DB PRINCIPAL".REFERENCIAS.PASSO_DEC)
      { S7_GenerateENO := "TRUE" } Move(in := "DB PRINCIPAL".REFERENCIAS.PASSO_DEC, out1 => "DB EXTRACTA2".REFERENCIAS.FINAL)
   END_RUNG
   // the same network as SCL:
   // ENO of a box is taken as its EN; it also drops when the box reports an error
   #_w1 := "DB PRINCIPAL".AUXILIARES.SEMPRE_1 AND %DB16.DBX4.5;
   IF #_w1 AND ("Tag_56" > "DB EXTRACTA2".REFERENCIAS.FINAL) THEN
       "DB EXTRACTA2".REFERENCIAS.FINAL := "DB EXTRACTA2".REFERENCIAS.FINAL + "DB PRINCIPAL".REFERENCIAS.PASSO_ACC;
   END_IF;
   #_w2 := #_w1 AND ("DB EXTRACTA2".REFERENCIAS.FINAL > "Tag_56");
   IF #_w2 THEN
       "DB EXTRACTA2".REFERENCIAS.FINAL := "DB EXTRACTA2".REFERENCIAS.FINAL - "DB PRINCIPAL".REFERENCIAS.PASSO_DEC;
   END_IF;
   IF #_w2 AND ("DB EXTRACTA2".REFERENCIAS.FINAL < 0.0) THEN "DB EXTRACTA2".REFERENCIAS.FINAL := 0.0; END_IF;
   IF #_w1 THEN "Tag_58" := "DB EXTRACTA2".REFERENCIAS.FINAL - "Tag_56"; END_IF;
   IF #_w1 AND ("Tag_58" > (-1.0)) AND ("Tag_58" < 1.0) THEN
       "DB EXTRACTA2".REFERENCIAS.FINAL := "Tag_56";
   END_IF;
   IF #_w1 AND NOT "DB EXTRACTA2".COMANDOS.DESBLOQUEIO_DRIVER AND ("DB EXTRACTA2".REFERENCIAS.FINAL >= "DB PRINCIPAL".REFERENCIAS.PASSO_DEC) THEN
       "DB EXTRACTA2".REFERENCIAS.FINAL := "DB PRINCIPAL".REFERENCIAS.PASSO_DEC;
   END_IF;
END_REGION

REGION Network 13
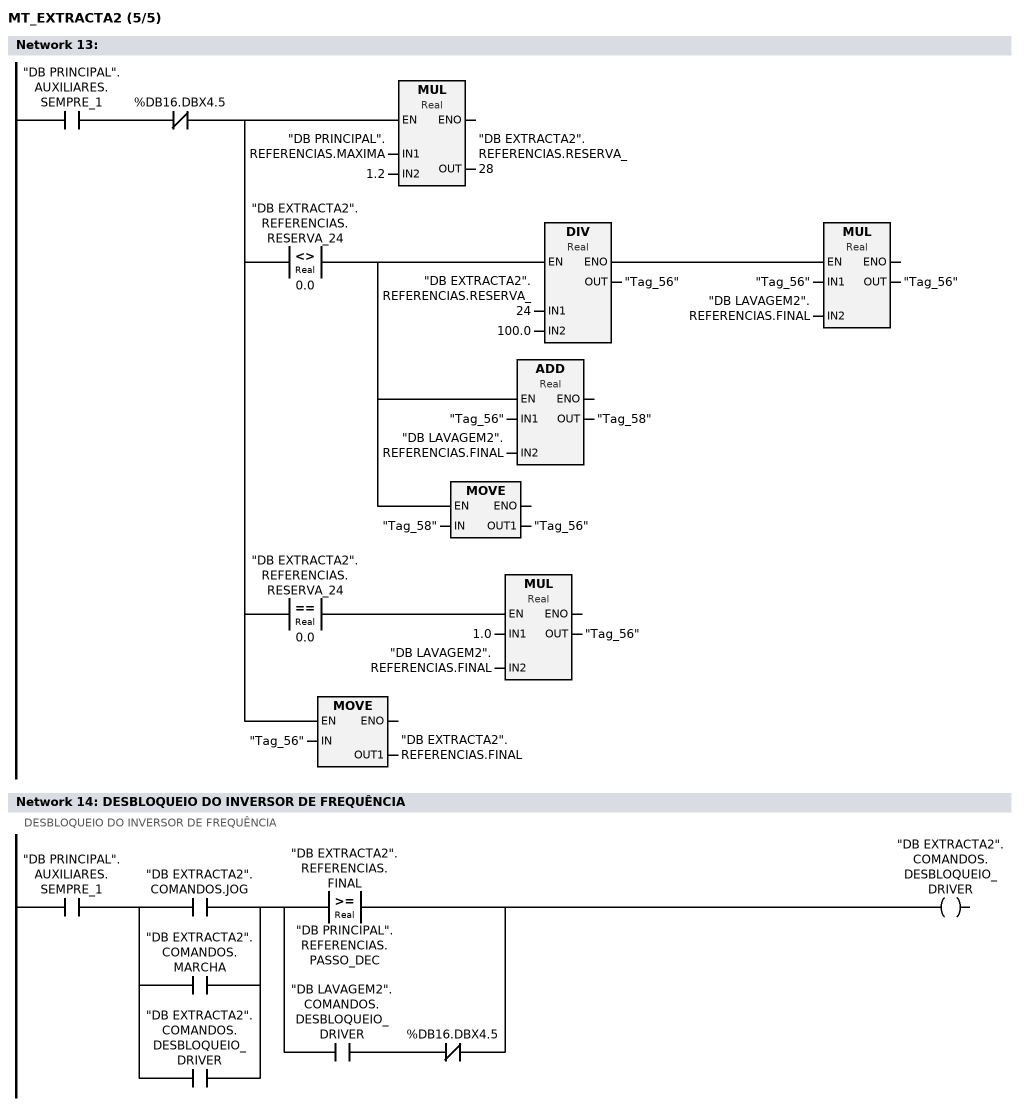
   RUNG wire#powerrail
      Contact( "DB PRINCIPAL".AUXILIARES.SEMPRE_1 )
      I_Contact( %DB16.DBX4.5 )
      wire#w1
      { S7_Templates := "SrcType := Real"; S7_GenerateENO := "TRUE" } Mul(in1 := "DB PRINCIPAL".REFERENCIAS.MAXIMA, in2 := 1.2, out => "DB EXTRACTA2".REFERENCIAS.RESERVA_28)
   END_RUNG
   RUNG wire#w1
      { S7_Templates := "SrcType := Real" } NE_Contact(in1 := "DB EXTRACTA2".REFERENCIAS.RESERVA_24, in2 := 0.0)
      wire#w2
      { S7_Templates := "SrcType := Real"; S7_GenerateENO := "TRUE" } Div(in1 := "DB EXTRACTA2".REFERENCIAS.RESERVA_24, in2 := 100.0, out => "Tag_56")
      { S7_Templates := "SrcType := Real"; S7_GenerateENO := "TRUE" } Mul(in1 := "Tag_56", in2 := "DB LAVAGEM2".REFERENCIAS.FINAL, out => "Tag_56")
   END_RUNG
   RUNG wire#w2
      { S7_Templates := "SrcType := Real"; S7_GenerateENO := "TRUE" } Add(in1 := "Tag_56", in2 := "DB LAVAGEM2".REFERENCIAS.FINAL, out => "Tag_58")
   END_RUNG
   RUNG wire#w2
      { S7_GenerateENO := "TRUE" } Move(in := "Tag_58", out1 => "Tag_56")
   END_RUNG
   RUNG wire#w1
      { S7_Templates := "SrcType := Real" } EQ_Contact(in1 := "DB EXTRACTA2".REFERENCIAS.RESERVA_24, in2 := 0.0)
      { S7_Templates := "SrcType := Real"; S7_GenerateENO := "TRUE" } Mul(in1 := 1.0, in2 := "DB LAVAGEM2".REFERENCIAS.FINAL, out => "Tag_56")
   END_RUNG
   RUNG wire#w1
      { S7_GenerateENO := "TRUE" } Move(in := "Tag_56", out1 => "DB EXTRACTA2".REFERENCIAS.FINAL)
   END_RUNG
   // the same network as SCL:
   // ENO of a box is taken as its EN; it also drops when the box reports an error
   #_w1 := "DB PRINCIPAL".AUXILIARES.SEMPRE_1 AND NOT %DB16.DBX4.5;
   IF #_w1 THEN "DB EXTRACTA2".REFERENCIAS.RESERVA_28 := "DB PRINCIPAL".REFERENCIAS.MAXIMA * 1.2; END_IF;
   IF #_w1 AND ("DB EXTRACTA2".REFERENCIAS.RESERVA_24 <> 0.0) THEN
       "Tag_56" := "DB EXTRACTA2".REFERENCIAS.RESERVA_24 / 100.0;
       "Tag_56" := "Tag_56" * "DB LAVAGEM2".REFERENCIAS.FINAL;
       "Tag_58" := "Tag_56" + "DB LAVAGEM2".REFERENCIAS.FINAL;
       "Tag_56" := "Tag_58";
   END_IF;
   IF #_w1 AND ("DB EXTRACTA2".REFERENCIAS.RESERVA_24 = 0.0) THEN
       "Tag_56" := 1.0 * "DB LAVAGEM2".REFERENCIAS.FINAL;
   END_IF;
   IF #_w1 THEN "DB EXTRACTA2".REFERENCIAS.FINAL := "Tag_56"; END_IF;
END_REGION

REGION Network 14: DESBLOQUEIO DO INVERSOR DE FREQUÊNCIA
   // DESBLOQUEIO DO INVERSOR DE FREQUÊNCIA
   RUNG wire#powerrail
      Contact( "DB PRINCIPAL".AUXILIARES.SEMPRE_1 )
      wire#w1
      Contact( "DB EXTRACTA2".COMANDOS.JOG )
      wire#w2
      { S7_Templates := "SrcType := Real" } GE_Contact(in1 := "DB EXTRACTA2".REFERENCIAS.FINAL, in2 := "DB PRINCIPAL".REFERENCIAS.PASSO_DEC)
      wire#w3
      Coil( "DB EXTRACTA2".COMANDOS.DESBLOQUEIO_DRIVER )
   END_RUNG
   RUNG wire#w1
      Contact( "DB EXTRACTA2".COMANDOS.MARCHA )
   END_RUNG wire#w2
   RUNG wire#w1
      Contact( "DB EXTRACTA2".COMANDOS.DESBLOQUEIO_DRIVER )
   END_RUNG wire#w2
   RUNG wire#w2
      Contact( "DB LAVAGEM2".COMANDOS.DESBLOQUEIO_DRIVER )
      I_Contact( %DB16.DBX4.5 )
   END_RUNG wire#w3
   // the same network as SCL:
   "DB EXTRACTA2".COMANDOS.DESBLOQUEIO_DRIVER := "DB PRINCIPAL".AUXILIARES.SEMPRE_1 AND ("DB EXTRACTA2".COMANDOS.JOG OR "DB EXTRACTA2".COMANDOS.MARCHA OR "DB EXTRACTA2".COMANDOS.DESBLOQUEIO_DRIVER) AND (("DB EXTRACTA2".REFERENCIAS.FINAL >= "DB PRINCIPAL".REFERENCIAS.PASSO_DEC) OR ("DB LAVAGEM2".COMANDOS.DESBLOQUEIO_DRIVER AND NOT %DB16.DBX4.5));
END_REGION

REGION Network 15 (STL): STATUS / CONTROLE - INVERSOR DE FREQUÊNCIA
   // DANFOSS FC300 PROFIBUS - TEX24626INV001
   // STATUS DO INVERSOR DE FREQUÊNCIA
         L     "Tag_17":P;
         T     "Tag_1";
         AN    "Tag_59";
         =     "DB EXTRACTA2".COMANDOS.STATUS_DRIVER;

   // CONTROLE DO INVERSOR DE FREQUÊNCIA
         L     1150;
         T     "Tag_1";
         A     "DB EXTRACTA2".COMANDOS.DESBLOQUEIO_DRIVER;
         =     "Tag_60";
         A     "T2";
         AN    "DB EXTRACTA2".COMANDOS.STATUS_DRIVER;
         =     "Tag_61";
         L     "Tag_1";
         T     "Tag_18":P;

   // REFERÊNCIA PARA O INVERSOR DE FREQUÊNCIA
         L     "DB EXTRACTA2".REFERENCIAS.FINAL;
         RND;
         T     "Tag_19":P;
END_REGION

REGION Network 16 (STL): INVERSOR RESERVA
         A     "DB PRINCIPAL".AUXILIARES.SEMPRE_1;
         =     %L24.0;
         A     %L24.0;
         A(;
         L     "DB PRINCIPAL".AUXILIARES1.INVERSOR_RESERVA1;
         L     7;
         ==I;
         );
         =     %L24.1;
         A     %L24.1;
         JNB   M00f;
         L     "DB EXTRACTA2".REFERENCIAS.FINAL;
         L     3.456;
         *R;
         T     #AUX_R;
         RND;
         T     "P_QW100":P;
   M00f: NOP   0;
         A     %L24.1;
         A     "I130";
         S     "DB PRINCIPAL".ALARME.INV_RESERVA1;
         A     %L24.1;
         A     "DB EXTRACTA2".COMANDOS.DESBLOQUEIO_DRIVER;
         S     "Q134";
         A     %L24.1;
         AN    "DB EXTRACTA2".COMANDOS.DESBLOQUEIO_DRIVER;
         R     "Q134";
         A     %L24.0;
         A(;
         L     "DB PRINCIPAL".AUXILIARES1.INVERSOR_RESERVA2;
         L     7;
         ==I;
         );
         =     %L24.1;
         A     %L24.1;
         JNB   M010;
         L     "DB EXTRACTA2".REFERENCIAS.FINAL;
         L     3.456;
         *R;
         T     #AUX_R;
         RND;
         T     "P_QW102":P;
   M010: NOP   0;
         A     %L24.1;
         A     "I132";
         S     "DB PRINCIPAL".ALARME.INV_RESERVA2;
         A     %L24.1;
         A     "DB EXTRACTA2".COMANDOS.DESBLOQUEIO_DRIVER;
         S     "Q135";
         A     %L24.1;
         AN    "DB EXTRACTA2".COMANDOS.DESBLOQUEIO_DRIVER;
         R     "Q135";
END_REGION
END_FUNCTION

FUNCTION "MT_LAVAGEM2" : Void   // FC17, LAD
TITLE = MÓDULO DE CONTROLE DA LAVAGEM 2
{ S7_Optimized_Access := 'FALSE' }
AUTHOR : THALLES
FAMILY : TRAÇÃO
NAME : LINHA1
VERSION : 0.1
// DATA BLOCK DE CONTROLE // DB17
// Automation Pack Automação Indl. e Com. Ltda.
// Cliente: Texima S/A Ind. de Máquinas
// Cliente Final: Cia. Fiação e Tecidos Santo Antonio.
// Máquina: LINHA 1 DENIN - O.S.: 24.626
   VAR_TEMP
      AUX_R : Real;
   END_VAR
   VAR_TEMP   // added for the SCL form of the ladder/FBD networks
      _w1 : Bool;
   END_VAR
BEGIN

REGION Network 1: ALARMES
   // RESET DOS ALARMES
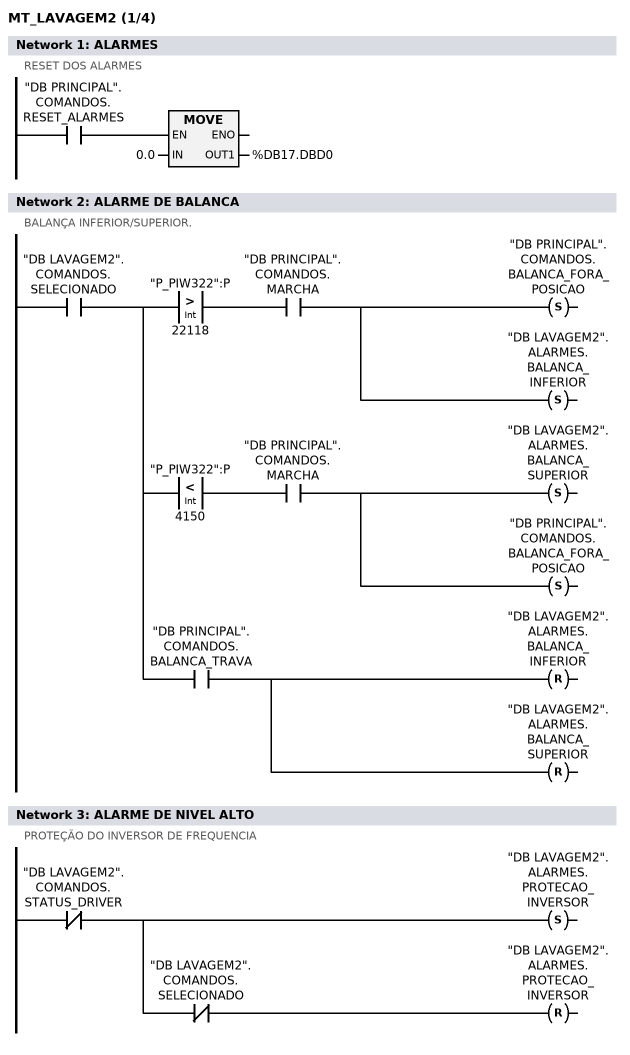
   RUNG wire#powerrail
      Contact( "DB PRINCIPAL".COMANDOS.RESET_ALARMES )
      { S7_GenerateENO := "TRUE" } Move(in := 0.0, out1 => %DB17.DBD0)
   END_RUNG
   // the same network as SCL:
   IF "DB PRINCIPAL".COMANDOS.RESET_ALARMES THEN %DB17.DBD0 := 0.0; END_IF;
END_REGION

REGION Network 2: ALARME DE BALANCA
   // BALANÇA INFERIOR/SUPERIOR.
   RUNG wire#powerrail
      Contact( "DB LAVAGEM2".COMANDOS.SELECIONADO )
      wire#w1
      { S7_Templates := "SrcType := Int" } GT_Contact(in1 := "P_PIW322":P, in2 := 22118)
      Contact( "DB PRINCIPAL".COMANDOS.MARCHA )
      wire#w2
      S_Coil( "DB PRINCIPAL".COMANDOS.BALANCA_FORA_POSICAO )
   END_RUNG
   RUNG wire#w2
      S_Coil( "DB LAVAGEM2".ALARMES.BALANCA_INFERIOR )
   END_RUNG
   RUNG wire#w1
      { S7_Templates := "SrcType := Int" } LT_Contact(in1 := "P_PIW322":P, in2 := 4150)
      Contact( "DB PRINCIPAL".COMANDOS.MARCHA )
      wire#w3
      S_Coil( "DB LAVAGEM2".ALARMES.BALANCA_SUPERIOR )
   END_RUNG
   RUNG wire#w3
      S_Coil( "DB PRINCIPAL".COMANDOS.BALANCA_FORA_POSICAO )
   END_RUNG
   RUNG wire#w1
      Contact( "DB PRINCIPAL".COMANDOS.BALANCA_TRAVA )
      wire#w4
      R_Coil( "DB LAVAGEM2".ALARMES.BALANCA_INFERIOR )
   END_RUNG
   RUNG wire#w4
      R_Coil( "DB LAVAGEM2".ALARMES.BALANCA_SUPERIOR )
   END_RUNG
   // the same network as SCL:
   IF "DB LAVAGEM2".COMANDOS.SELECIONADO AND ("P_PIW322":P > 22118) AND "DB PRINCIPAL".COMANDOS.MARCHA THEN
       "DB PRINCIPAL".COMANDOS.BALANCA_FORA_POSICAO := TRUE;
       "DB LAVAGEM2".ALARMES.BALANCA_INFERIOR := TRUE;
   END_IF;
   IF "DB LAVAGEM2".COMANDOS.SELECIONADO AND ("P_PIW322":P < 4150) AND "DB PRINCIPAL".COMANDOS.MARCHA THEN
       "DB LAVAGEM2".ALARMES.BALANCA_SUPERIOR := TRUE;
       "DB PRINCIPAL".COMANDOS.BALANCA_FORA_POSICAO := TRUE;
   END_IF;
   IF "DB LAVAGEM2".COMANDOS.SELECIONADO AND "DB PRINCIPAL".COMANDOS.BALANCA_TRAVA THEN
       "DB LAVAGEM2".ALARMES.BALANCA_INFERIOR := FALSE;
       "DB LAVAGEM2".ALARMES.BALANCA_SUPERIOR := FALSE;
   END_IF;
END_REGION

REGION Network 3: ALARME DE NIVEL ALTO
   // PROTEÇÃO DO INVERSOR DE FREQUENCIA
   RUNG wire#powerrail
      I_Contact( "DB LAVAGEM2".COMANDOS.STATUS_DRIVER )
      wire#w1
      S_Coil( "DB LAVAGEM2".ALARMES.PROTECAO_INVERSOR )
   END_RUNG
   RUNG wire#w1
      I_Contact( "DB LAVAGEM2".COMANDOS.SELECIONADO )
      R_Coil( "DB LAVAGEM2".ALARMES.PROTECAO_INVERSOR )
   END_RUNG
   // the same network as SCL:
   #_w1 := NOT "DB LAVAGEM2".COMANDOS.STATUS_DRIVER;
   IF #_w1 THEN "DB LAVAGEM2".ALARMES.PROTECAO_INVERSOR := TRUE; END_IF;
   IF #_w1 AND NOT "DB LAVAGEM2".COMANDOS.SELECIONADO THEN
       "DB LAVAGEM2".ALARMES.PROTECAO_INVERSOR := FALSE;
   END_IF;
END_REGION

REGION Network 4: ALARMES
   // ATIVAÇÃO DO BIT DE ALARME DE NIVEL ALTO
   // ATIVAÇÃO DO BIT DE ALARME DE NIVEL BAIXO
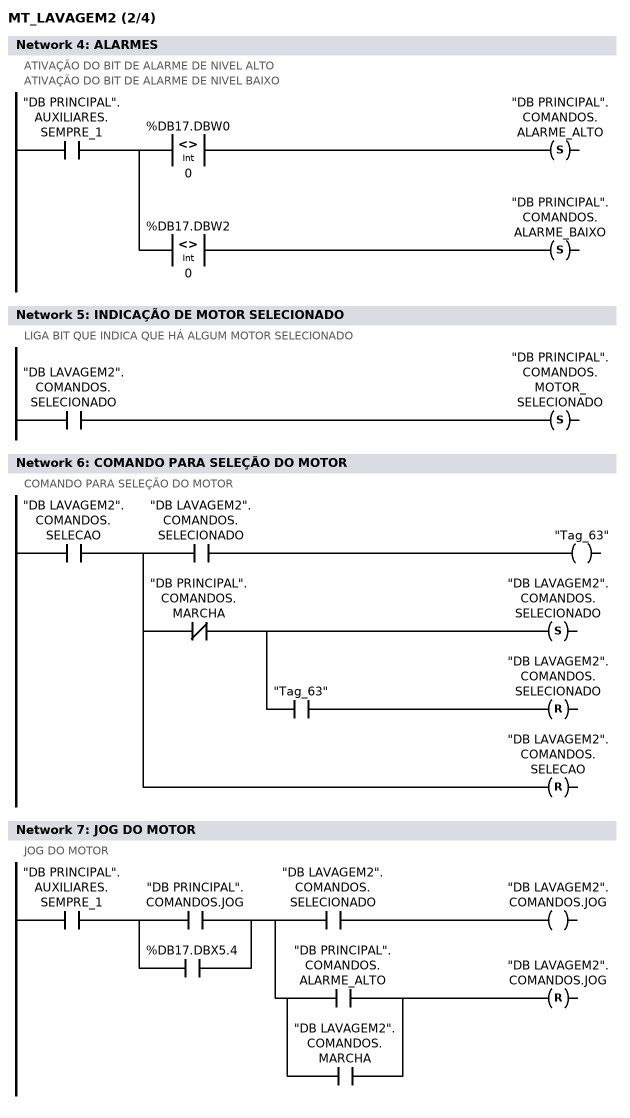
   RUNG wire#powerrail
      Contact( "DB PRINCIPAL".AUXILIARES.SEMPRE_1 )
      wire#w1
      { S7_Templates := "SrcType := Int" } NE_Contact(in1 := %DB17.DBW0, in2 := 0)
      S_Coil( "DB PRINCIPAL".COMANDOS.ALARME_ALTO )
   END_RUNG
   RUNG wire#w1
      { S7_Templates := "SrcType := Int" } NE_Contact(in1 := %DB17.DBW2, in2 := 0)
      S_Coil( "DB PRINCIPAL".COMANDOS.ALARME_BAIXO )
   END_RUNG
   // the same network as SCL:
   IF "DB PRINCIPAL".AUXILIARES.SEMPRE_1 AND (%DB17.DBW0 <> 0) THEN
       "DB PRINCIPAL".COMANDOS.ALARME_ALTO := TRUE;
   END_IF;
   IF "DB PRINCIPAL".AUXILIARES.SEMPRE_1 AND (%DB17.DBW2 <> 0) THEN
       "DB PRINCIPAL".COMANDOS.ALARME_BAIXO := TRUE;
   END_IF;
END_REGION

REGION Network 5: INDICAÇÃO DE MOTOR SELECIONADO
   // LIGA BIT QUE INDICA QUE HÁ ALGUM MOTOR SELECIONADO
   RUNG wire#powerrail
      Contact( "DB LAVAGEM2".COMANDOS.SELECIONADO )
      S_Coil( "DB PRINCIPAL".COMANDOS.MOTOR_SELECIONADO )
   END_RUNG
   // the same network as SCL:
   IF "DB LAVAGEM2".COMANDOS.SELECIONADO THEN "DB PRINCIPAL".COMANDOS.MOTOR_SELECIONADO := TRUE; END_IF;
END_REGION

REGION Network 6: COMANDO PARA SELEÇÃO DO MOTOR
   // COMANDO PARA SELEÇÃO DO MOTOR
   RUNG wire#powerrail
      Contact( "DB LAVAGEM2".COMANDOS.SELECAO )
      wire#w1
      Contact( "DB LAVAGEM2".COMANDOS.SELECIONADO )
      Coil( "Tag_63" )
   END_RUNG
   RUNG wire#w1
      I_Contact( "DB PRINCIPAL".COMANDOS.MARCHA )
      wire#w2
      S_Coil( "DB LAVAGEM2".COMANDOS.SELECIONADO )
   END_RUNG
   RUNG wire#w2
      Contact( "Tag_63" )
      R_Coil( "DB LAVAGEM2".COMANDOS.SELECIONADO )
   END_RUNG
   RUNG wire#w1
      R_Coil( "DB LAVAGEM2".COMANDOS.SELECAO )
   END_RUNG
   // the same network as SCL:
   "Tag_63" := "DB LAVAGEM2".COMANDOS.SELECAO AND "DB LAVAGEM2".COMANDOS.SELECIONADO;
   #_w1 := "DB LAVAGEM2".COMANDOS.SELECAO AND NOT "DB PRINCIPAL".COMANDOS.MARCHA;
   IF #_w1 THEN "DB LAVAGEM2".COMANDOS.SELECIONADO := TRUE; END_IF;
   IF #_w1 AND "Tag_63" THEN "DB LAVAGEM2".COMANDOS.SELECIONADO := FALSE; END_IF;
   IF "DB LAVAGEM2".COMANDOS.SELECAO THEN "DB LAVAGEM2".COMANDOS.SELECAO := FALSE; END_IF;
END_REGION

REGION Network 7: JOG DO MOTOR
   // JOG DO MOTOR
   RUNG wire#powerrail
      Contact( "DB PRINCIPAL".AUXILIARES.SEMPRE_1 )
      wire#w1
      Contact( "DB PRINCIPAL".COMANDOS.JOG )
      wire#w2
      Contact( "DB LAVAGEM2".COMANDOS.SELECIONADO )
      Coil( "DB LAVAGEM2".COMANDOS.JOG )
   END_RUNG
   RUNG wire#w1
      Contact( %DB17.DBX5.4 )
   END_RUNG wire#w2
   RUNG wire#w2
      Contact( "DB PRINCIPAL".COMANDOS.ALARME_ALTO )
      wire#w3
      R_Coil( "DB LAVAGEM2".COMANDOS.JOG )
   END_RUNG
   RUNG wire#w2
      Contact( "DB LAVAGEM2".COMANDOS.MARCHA )
   END_RUNG wire#w3
   // the same network as SCL:
   #_w1 := "DB PRINCIPAL".AUXILIARES.SEMPRE_1 AND ("DB PRINCIPAL".COMANDOS.JOG OR %DB17.DBX5.4);
   "DB LAVAGEM2".COMANDOS.JOG := #_w1 AND "DB LAVAGEM2".COMANDOS.SELECIONADO;
   IF #_w1 AND ("DB PRINCIPAL".COMANDOS.ALARME_ALTO OR "DB LAVAGEM2".COMANDOS.MARCHA) THEN
       "DB LAVAGEM2".COMANDOS.JOG := FALSE;
   END_IF;
END_REGION

REGION Network 8: COMANDO PARA LIBERAÇÃO DO MOTOR
   // COMANDO PARA LIBERAÇÃO DO MOTOR
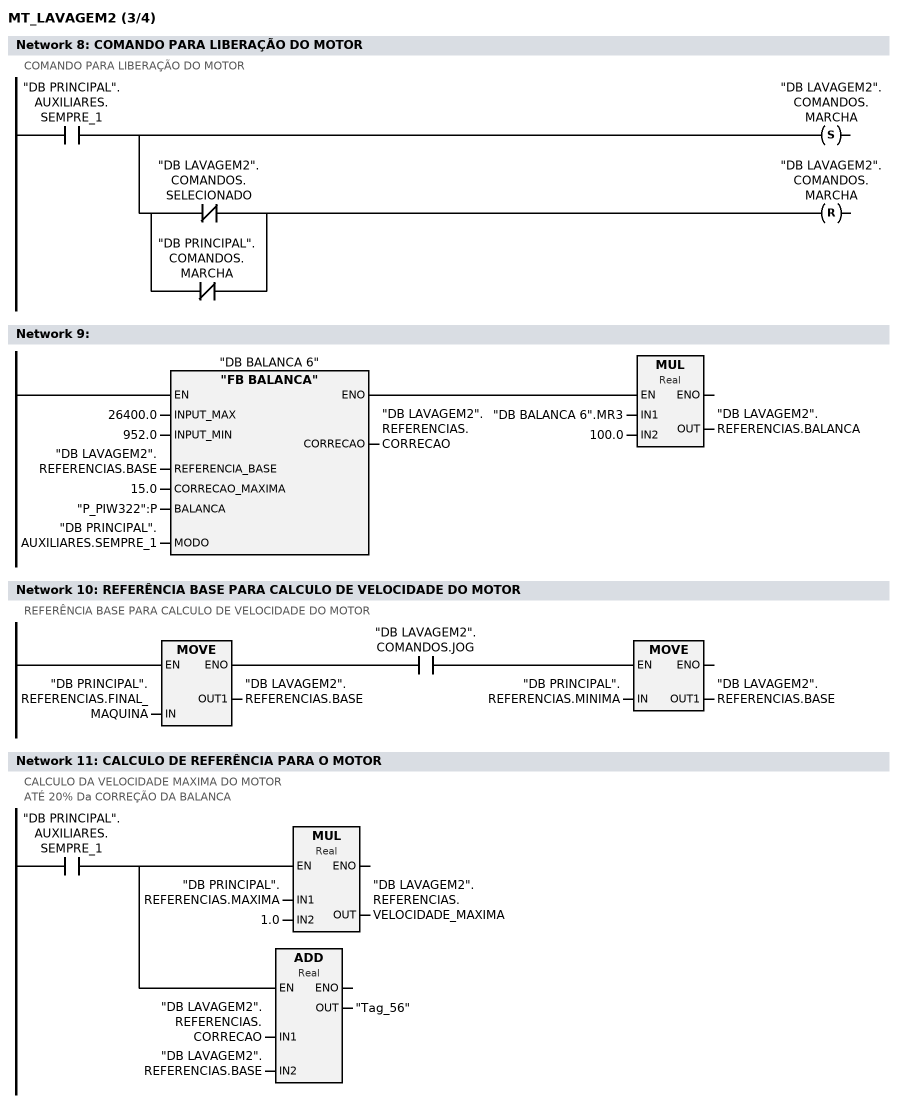
   RUNG wire#powerrail
      Contact( "DB PRINCIPAL".AUXILIARES.SEMPRE_1 )
      wire#w1
      S_Coil( "DB LAVAGEM2".COMANDOS.MARCHA )
   END_RUNG
   RUNG wire#w1
      I_Contact( "DB LAVAGEM2".COMANDOS.SELECIONADO )
      wire#w2
      R_Coil( "DB LAVAGEM2".COMANDOS.MARCHA )
   END_RUNG
   RUNG wire#w1
      I_Contact( "DB PRINCIPAL".COMANDOS.MARCHA )
   END_RUNG wire#w2
   // the same network as SCL:
   IF "DB PRINCIPAL".AUXILIARES.SEMPRE_1 THEN "DB LAVAGEM2".COMANDOS.MARCHA := TRUE; END_IF;
   IF "DB PRINCIPAL".AUXILIARES.SEMPRE_1 AND (NOT "DB LAVAGEM2".COMANDOS.SELECIONADO OR NOT "DB PRINCIPAL".COMANDOS.MARCHA) THEN
       "DB LAVAGEM2".COMANDOS.MARCHA := FALSE;
   END_IF;
END_REGION

REGION Network 9
   RUNG wire#powerrail
      "DB BALANCA 6"(INPUT_MAX := 26400.0, INPUT_MIN := 952.0, REFERENCIA_BASE := "DB LAVAGEM2".REFERENCIAS.BASE, CORRECAO_MAXIMA := 15.0, BALANCA := "P_PIW322":P, MODO := "DB PRINCIPAL".AUXILIARES.SEMPRE_1, CORRECAO => "DB LAVAGEM2".REFERENCIAS.CORRECAO)
      { S7_Templates := "SrcType := Real"; S7_GenerateENO := "TRUE" } Mul(in1 := "DB BALANCA 6".MR3, in2 := 100.0, out => "DB LAVAGEM2".REFERENCIAS.BALANCA)
   END_RUNG
   // the same network as SCL:
   "DB BALANCA 6"(INPUT_MAX := 26400.0,   // "FB BALANCA"
                  INPUT_MIN := 952.0,
                  REFERENCIA_BASE := "DB LAVAGEM2".REFERENCIAS.BASE,
                  CORRECAO_MAXIMA := 15.0,
                  BALANCA := "P_PIW322":P,
                  MODO := "DB PRINCIPAL".AUXILIARES.SEMPRE_1,
                  CORRECAO => "DB LAVAGEM2".REFERENCIAS.CORRECAO,
                  ENO => #_w1);
   IF #_w1 THEN "DB LAVAGEM2".REFERENCIAS.BALANCA := "DB BALANCA 6".MR3 * 100.0; END_IF;
END_REGION

REGION Network 10: REFERÊNCIA BASE PARA CALCULO DE VELOCIDADE DO MOTOR
   // REFERÊNCIA BASE PARA CALCULO DE VELOCIDADE DO MOTOR
   RUNG wire#powerrail
      { S7_GenerateENO := "TRUE" } Move(in := "DB PRINCIPAL".REFERENCIAS.FINAL_MAQUINA, out1 => "DB LAVAGEM2".REFERENCIAS.BASE)
      Contact( "DB LAVAGEM2".COMANDOS.JOG )
      { S7_GenerateENO := "TRUE" } Move(in := "DB PRINCIPAL".REFERENCIAS.MINIMA, out1 => "DB LAVAGEM2".REFERENCIAS.BASE)
   END_RUNG
   // the same network as SCL:
   // ENO of a box is taken as its EN; it also drops when the box reports an error
   "DB LAVAGEM2".REFERENCIAS.BASE := "DB PRINCIPAL".REFERENCIAS.FINAL_MAQUINA;
   IF "DB LAVAGEM2".COMANDOS.JOG THEN
       "DB LAVAGEM2".REFERENCIAS.BASE := "DB PRINCIPAL".REFERENCIAS.MINIMA;
   END_IF;
END_REGION

REGION Network 11: CALCULO DE REFERÊNCIA PARA O MOTOR
   // CALCULO DA VELOCIDADE MAXIMA DO MOTOR
   // ATÉ 20% Da CORREÇÃO DA BALANCA
   RUNG wire#powerrail
      Contact( "DB PRINCIPAL".AUXILIARES.SEMPRE_1 )
      wire#w1
      { S7_Templates := "SrcType := Real"; S7_GenerateENO := "TRUE" } Mul(in1 := "DB PRINCIPAL".REFERENCIAS.MAXIMA, in2 := 1.0, out => "DB LAVAGEM2".REFERENCIAS.VELOCIDADE_MAXIMA)
   END_RUNG
   RUNG wire#w1
      { S7_Templates := "SrcType := Real"; S7_GenerateENO := "TRUE" } Add(in1 := "DB LAVAGEM2".REFERENCIAS.CORRECAO, in2 := "DB LAVAGEM2".REFERENCIAS.BASE, out => "Tag_56")
   END_RUNG
   // the same network as SCL:
   IF "DB PRINCIPAL".AUXILIARES.SEMPRE_1 THEN
       "DB LAVAGEM2".REFERENCIAS.VELOCIDADE_MAXIMA := "DB PRINCIPAL".REFERENCIAS.MAXIMA * 1.0;
       "Tag_56" := "DB LAVAGEM2".REFERENCIAS.CORRECAO + "DB LAVAGEM2".REFERENCIAS.BASE;
   END_IF;
END_REGION

REGION Network 12: ACC/DEC DA REFERÊNCIA DO MOTOR
   // ACC/DEC DA REFERÊNCIA DO MOTOR
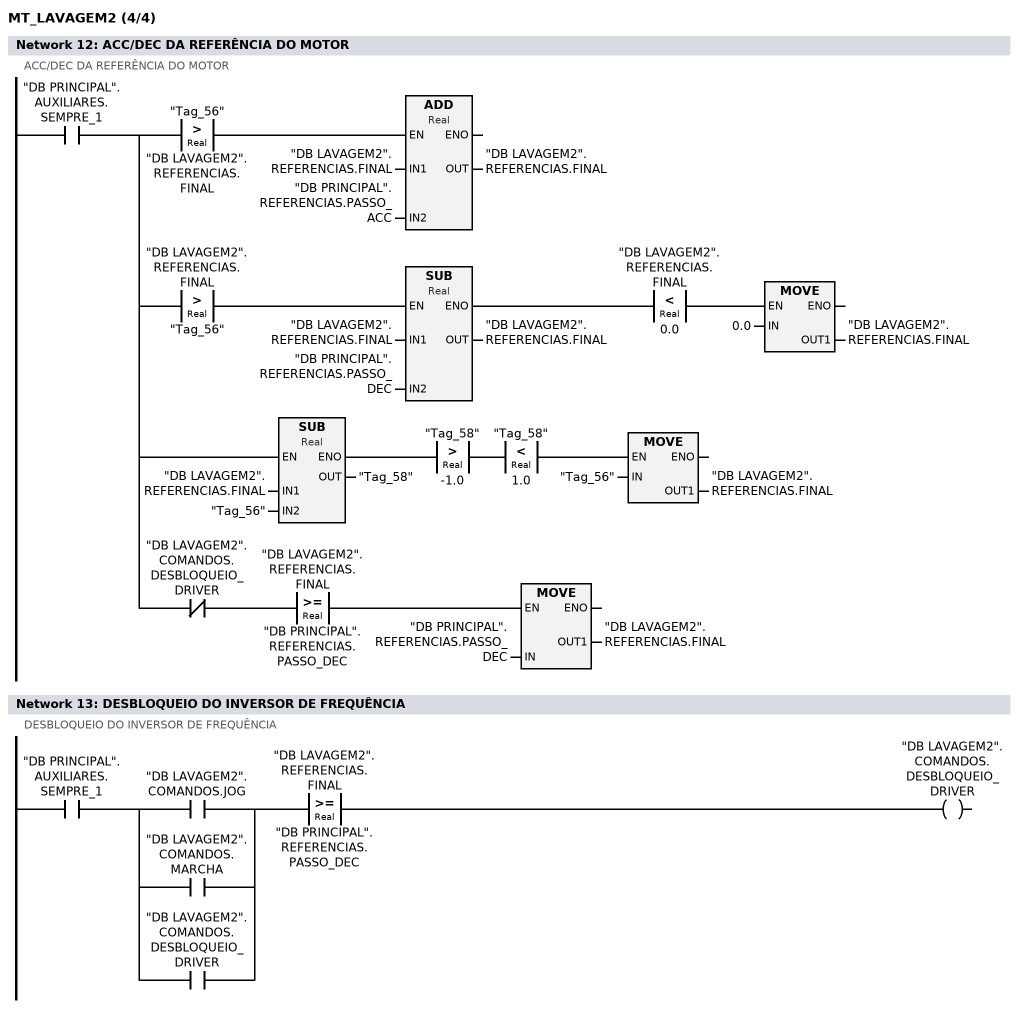
   RUNG wire#powerrail
      Contact( "DB PRINCIPAL".AUXILIARES.SEMPRE_1 )
      wire#w1
      { S7_Templates := "SrcType := Real" } GT_Contact(in1 := "Tag_56", in2 := "DB LAVAGEM2".REFERENCIAS.FINAL)
      { S7_Templates := "SrcType := Real"; S7_GenerateENO := "TRUE" } Add(in1 := "DB LAVAGEM2".REFERENCIAS.FINAL, in2 := "DB PRINCIPAL".REFERENCIAS.PASSO_ACC, out => "DB LAVAGEM2".REFERENCIAS.FINAL)
   END_RUNG
   RUNG wire#w1
      { S7_Templates := "SrcType := Real" } GT_Contact(in1 := "DB LAVAGEM2".REFERENCIAS.FINAL, in2 := "Tag_56")
      { S7_Templates := "SrcType := Real"; S7_GenerateENO := "TRUE" } Sub(in1 := "DB LAVAGEM2".REFERENCIAS.FINAL, in2 := "DB PRINCIPAL".REFERENCIAS.PASSO_DEC, out => "DB LAVAGEM2".REFERENCIAS.FINAL)
      { S7_Templates := "SrcType := Real" } LT_Contact(in1 := "DB LAVAGEM2".REFERENCIAS.FINAL, in2 := 0.0)
      { S7_GenerateENO := "TRUE" } Move(in := 0.0, out1 => "DB LAVAGEM2".REFERENCIAS.FINAL)
   END_RUNG
   RUNG wire#w1
      { S7_Templates := "SrcType := Real"; S7_GenerateENO := "TRUE" } Sub(in1 := "DB LAVAGEM2".REFERENCIAS.FINAL, in2 := "Tag_56", out => "Tag_58")
      { S7_Templates := "SrcType := Real" } GT_Contact(in1 := "Tag_58", in2 := -1.0)
      { S7_Templates := "SrcType := Real" } LT_Contact(in1 := "Tag_58", in2 := 1.0)
      { S7_GenerateENO := "TRUE" } Move(in := "Tag_56", out1 => "DB LAVAGEM2".REFERENCIAS.FINAL)
   END_RUNG
   RUNG wire#w1
      I_Contact( "DB LAVAGEM2".COMANDOS.DESBLOQUEIO_DRIVER )
      { S7_Templates := "SrcType := Real" } GE_Contact(in1 := "DB LAVAGEM2".REFERENCIAS.FINAL, in2 := "DB PRINCIPAL".REFERENCIAS.PASSO_DEC)
      { S7_GenerateENO := "TRUE" } Move(in := "DB PRINCIPAL".REFERENCIAS.PASSO_DEC, out1 => "DB LAVAGEM2".REFERENCIAS.FINAL)
   END_RUNG
   // the same network as SCL:
   // ENO of a box is taken as its EN; it also drops when the box reports an error
   IF "DB PRINCIPAL".AUXILIARES.SEMPRE_1 AND ("Tag_56" > "DB LAVAGEM2".REFERENCIAS.FINAL) THEN
       "DB LAVAGEM2".REFERENCIAS.FINAL := "DB LAVAGEM2".REFERENCIAS.FINAL + "DB PRINCIPAL".REFERENCIAS.PASSO_ACC;
   END_IF;
   #_w1 := "DB PRINCIPAL".AUXILIARES.SEMPRE_1 AND ("DB LAVAGEM2".REFERENCIAS.FINAL > "Tag_56");
   IF #_w1 THEN
       "DB LAVAGEM2".REFERENCIAS.FINAL := "DB LAVAGEM2".REFERENCIAS.FINAL - "DB PRINCIPAL".REFERENCIAS.PASSO_DEC;
   END_IF;
   IF #_w1 AND ("DB LAVAGEM2".REFERENCIAS.FINAL < 0.0) THEN "DB LAVAGEM2".REFERENCIAS.FINAL := 0.0; END_IF;
   IF "DB PRINCIPAL".AUXILIARES.SEMPRE_1 THEN "Tag_58" := "DB LAVAGEM2".REFERENCIAS.FINAL - "Tag_56"; END_IF;
   IF "DB PRINCIPAL".AUXILIARES.SEMPRE_1 AND ("Tag_58" > (-1.0)) AND ("Tag_58" < 1.0) THEN
       "DB LAVAGEM2".REFERENCIAS.FINAL := "Tag_56";
   END_IF;
   IF "DB PRINCIPAL".AUXILIARES.SEMPRE_1 AND NOT "DB LAVAGEM2".COMANDOS.DESBLOQUEIO_DRIVER AND ("DB LAVAGEM2".REFERENCIAS.FINAL >= "DB PRINCIPAL".REFERENCIAS.PASSO_DEC) THEN
       "DB LAVAGEM2".REFERENCIAS.FINAL := "DB PRINCIPAL".REFERENCIAS.PASSO_DEC;
   END_IF;
END_REGION

REGION Network 13: DESBLOQUEIO DO INVERSOR DE FREQUÊNCIA
   // DESBLOQUEIO DO INVERSOR DE FREQUÊNCIA
   RUNG wire#powerrail
      Contact( "DB PRINCIPAL".AUXILIARES.SEMPRE_1 )
      wire#w1
      Contact( "DB LAVAGEM2".COMANDOS.JOG )
      wire#w2
      { S7_Templates := "SrcType := Real" } GE_Contact(in1 := "DB LAVAGEM2".REFERENCIAS.FINAL, in2 := "DB PRINCIPAL".REFERENCIAS.PASSO_DEC)
      Coil( "DB LAVAGEM2".COMANDOS.DESBLOQUEIO_DRIVER )
   END_RUNG
   RUNG wire#w1
      Contact( "DB LAVAGEM2".COMANDOS.MARCHA )
   END_RUNG wire#w2
   RUNG wire#w1
      Contact( "DB LAVAGEM2".COMANDOS.DESBLOQUEIO_DRIVER )
   END_RUNG wire#w2
   // the same network as SCL:
   "DB LAVAGEM2".COMANDOS.DESBLOQUEIO_DRIVER := "DB PRINCIPAL".AUXILIARES.SEMPRE_1 AND ("DB LAVAGEM2".COMANDOS.JOG OR "DB LAVAGEM2".COMANDOS.MARCHA OR "DB LAVAGEM2".COMANDOS.DESBLOQUEIO_DRIVER) AND ("DB LAVAGEM2".REFERENCIAS.FINAL >= "DB PRINCIPAL".REFERENCIAS.PASSO_DEC);
END_REGION

REGION Network 14 (STL): STATUS / CONTROLE - INVERSOR DE FREQUÊNCIA
   // DANFOSS FC300 PROFIBUS - TEX24626INV001
   // STATUS DO INVERSOR DE FREQUÊNCIA
         L     "Tag_20":P;
         T     "Tag_1";
         AN    "Tag_59";
         =     "DB LAVAGEM2".COMANDOS.STATUS_DRIVER;

   // CONTROLE DO INVERSOR DE FREQUÊNCIA
         L     1150;
         T     "Tag_1";
         A     "DB LAVAGEM2".COMANDOS.DESBLOQUEIO_DRIVER;
         =     "Tag_60";
         A     "T2";
         AN    "DB LAVAGEM2".COMANDOS.STATUS_DRIVER;
         =     "Tag_61";
         L     "Tag_1";
         T     "Tag_21":P;

   // REFERÊNCIA PARA O INVERSOR DE FREQUÊNCIA
         L     "DB LAVAGEM2".REFERENCIAS.FINAL;
         L     16384.0;
         *R;

         L     "DB LAVAGEM2".REFERENCIAS.VELOCIDADE_MAXIMA;
         /R;
         RND;
         T     "Tag_62";
         L     "Tag_62";
         T     "Tag_22":P;
END_REGION

REGION Network 15 (STL): INVERSOR RESERVA
         A     "DB PRINCIPAL".AUXILIARES.SEMPRE_1;
         =     %L24.0;
         A     %L24.0;
         A(;
         L     "DB PRINCIPAL".AUXILIARES1.INVERSOR_RESERVA1;
         L     8;
         ==I;
         );
         =     %L24.1;
         A     %L24.1;
         JNB   M001;
         L     "DB LAVAGEM2".REFERENCIAS.FINAL;
         L     3.456;
         *R;
         T     #AUX_R;
         RND;
         T     "P_QW100":P;
   M001: NOP   0;
         A     %L24.1;
         A     "I130";
         S     "DB PRINCIPAL".ALARME.INV_RESERVA1;
         A     %L24.1;
         A     "DB LAVAGEM2".COMANDOS.DESBLOQUEIO_DRIVER;
         S     "Q134";
         A     %L24.1;
         AN    "DB LAVAGEM2".COMANDOS.DESBLOQUEIO_DRIVER;
         R     "Q134";
         A     %L24.0;
         A(;
         L     "DB PRINCIPAL".AUXILIARES1.INVERSOR_RESERVA2;
         L     8;
         ==I;
         );
         =     %L24.1;
         A     %L24.1;
         JNB   M002;
         L     "DB LAVAGEM2".REFERENCIAS.FINAL;
         L     3.456;
         *R;
         T     #AUX_R;
         RND;
         T     "P_QW102":P;
   M002: NOP   0;
         A     %L24.1;
         A     "I132";
         S     "DB PRINCIPAL".ALARME.INV_RESERVA2;
         A     %L24.1;
         A     "DB LAVAGEM2".COMANDOS.DESBLOQUEIO_DRIVER;
         S     "Q135";
         A     %L24.1;
         AN    "DB LAVAGEM2".COMANDOS.DESBLOQUEIO_DRIVER;
         R     "Q135";
END_REGION
END_FUNCTION

FUNCTION "MT_SECADEIRA1" : Void   // FC18, LAD
TITLE = MÓDULO DE CONTROLE DA SECADEIRA 1
{ S7_Optimized_Access := 'FALSE' }
AUTHOR : THALLES
FAMILY : TRAÇÃO
NAME : LINHA1
VERSION : 0.1
// DATA BLOCK DE CONTROLE // DB18
// Automation Pack Automação Indl. e Com. Ltda.
// Cliente: Texima S/A Ind. de Máquinas
// Cliente Final: Cia. Fiação e Tecidos Santo Antonio.
// Máquina: LINHA 1 DENIN - O.S.: 24.626
   VAR_TEMP
      AUX_R : Real;
   END_VAR
   VAR_TEMP   // added for the SCL form of the ladder/FBD networks
      _w1 : Bool;
   END_VAR
BEGIN

REGION Network 1: ALARMES
   // RESET DOS ALARMES
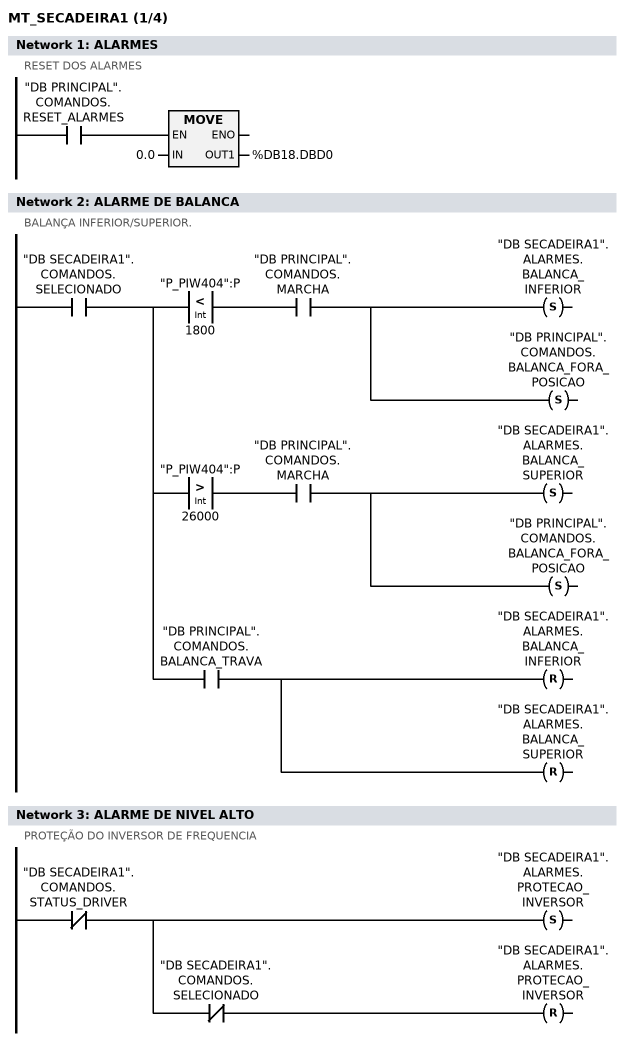
   RUNG wire#powerrail
      Contact( "DB PRINCIPAL".COMANDOS.RESET_ALARMES )
      { S7_GenerateENO := "TRUE" } Move(in := 0.0, out1 => %DB18.DBD0)
   END_RUNG
   // the same network as SCL:
   IF "DB PRINCIPAL".COMANDOS.RESET_ALARMES THEN %DB18.DBD0 := 0.0; END_IF;
END_REGION

REGION Network 2: ALARME DE BALANCA
   // BALANÇA INFERIOR/SUPERIOR.
   RUNG wire#powerrail
      Contact( "DB SECADEIRA1".COMANDOS.SELECIONADO )
      wire#w1
      { S7_Templates := "SrcType := Int" } LT_Contact(in1 := "P_PIW404":P, in2 := 1800)
      Contact( "DB PRINCIPAL".COMANDOS.MARCHA )
      wire#w2
      S_Coil( "DB SECADEIRA1".ALARMES.BALANCA_INFERIOR )
   END_RUNG
   RUNG wire#w2
      S_Coil( "DB PRINCIPAL".COMANDOS.BALANCA_FORA_POSICAO )
   END_RUNG
   RUNG wire#w1
      { S7_Templates := "SrcType := Int" } GT_Contact(in1 := "P_PIW404":P, in2 := 26000)
      Contact( "DB PRINCIPAL".COMANDOS.MARCHA )
      wire#w3
      S_Coil( "DB SECADEIRA1".ALARMES.BALANCA_SUPERIOR )
   END_RUNG
   RUNG wire#w3
      S_Coil( "DB PRINCIPAL".COMANDOS.BALANCA_FORA_POSICAO )
   END_RUNG
   RUNG wire#w1
      Contact( "DB PRINCIPAL".COMANDOS.BALANCA_TRAVA )
      wire#w4
      R_Coil( "DB SECADEIRA1".ALARMES.BALANCA_INFERIOR )
   END_RUNG
   RUNG wire#w4
      R_Coil( "DB SECADEIRA1".ALARMES.BALANCA_SUPERIOR )
   END_RUNG
   // the same network as SCL:
   IF "DB SECADEIRA1".COMANDOS.SELECIONADO AND ("P_PIW404":P < 1800) AND "DB PRINCIPAL".COMANDOS.MARCHA THEN
       "DB SECADEIRA1".ALARMES.BALANCA_INFERIOR := TRUE;
       "DB PRINCIPAL".COMANDOS.BALANCA_FORA_POSICAO := TRUE;
   END_IF;
   IF "DB SECADEIRA1".COMANDOS.SELECIONADO AND ("P_PIW404":P > 26000) AND "DB PRINCIPAL".COMANDOS.MARCHA THEN
       "DB SECADEIRA1".ALARMES.BALANCA_SUPERIOR := TRUE;
       "DB PRINCIPAL".COMANDOS.BALANCA_FORA_POSICAO := TRUE;
   END_IF;
   IF "DB SECADEIRA1".COMANDOS.SELECIONADO AND "DB PRINCIPAL".COMANDOS.BALANCA_TRAVA THEN
       "DB SECADEIRA1".ALARMES.BALANCA_INFERIOR := FALSE;
       "DB SECADEIRA1".ALARMES.BALANCA_SUPERIOR := FALSE;
   END_IF;
END_REGION

REGION Network 3: ALARME DE NIVEL ALTO
   // PROTEÇÃO DO INVERSOR DE FREQUENCIA
   RUNG wire#powerrail
      I_Contact( "DB SECADEIRA1".COMANDOS.STATUS_DRIVER )
      wire#w1
      S_Coil( "DB SECADEIRA1".ALARMES.PROTECAO_INVERSOR )
   END_RUNG
   RUNG wire#w1
      I_Contact( "DB SECADEIRA1".COMANDOS.SELECIONADO )
      R_Coil( "DB SECADEIRA1".ALARMES.PROTECAO_INVERSOR )
   END_RUNG
   // the same network as SCL:
   #_w1 := NOT "DB SECADEIRA1".COMANDOS.STATUS_DRIVER;
   IF #_w1 THEN "DB SECADEIRA1".ALARMES.PROTECAO_INVERSOR := TRUE; END_IF;
   IF #_w1 AND NOT "DB SECADEIRA1".COMANDOS.SELECIONADO THEN
       "DB SECADEIRA1".ALARMES.PROTECAO_INVERSOR := FALSE;
   END_IF;
END_REGION

REGION Network 4: ALARMES
   // ATIVAÇÃO DO BIT DE ALARME DE NIVEL ALTO
   // ATIVAÇÃO DO BIT DE ALARME DE NIVEL BAIXO
